LIN {X 0,Y 517.007,Z 176.899,A -85,B 0,C 180,E1 -4953.117,E2 -4953.117} C_VEL
LIN {X 0,Y 517.003,Z 176.9,A -85,B 0,C 180,E1 -4956.243,E2 -4956.243} C_VEL
LIN {X 0,Y 516.949,Z 176.905,A -85,B 0,C 180,E1 -4959.389,E2 -4959.389} C_VEL
LIN {X 0,Y 516.942,Z 176.905,A -85,B 0,C 180,E1 -4961.807,E2 -4961.807} C_VEL
LIN {X 0,Y 516.719,Z 176.937,A -85,B 0,C 180,E1 -4964.171,E2 -4964.171} C_VEL
LIN {X 0,Y 516.698,Z 177.952,A -85,B 0,C 180,E1 -4965.049,E2 -4965.049} C_VEL
LIN {X 0,Y 516.599,Z 183.078,A -85,B 0,C 180,E1 -4968.234,E2 -4968.234} C_VEL
LIN {X 0,Y 516.547,Z 187.118,A -85,B 0,C 180,E1 -4970.717,E2 -4970.717} C_VEL
LIN {X 0,Y 516.494,Z 191.277,A -85,B 0,C 180,E1 -4973.241,E2 -4973.241} C_VEL
LIN {X 0,Y 516.447,Z 196.01,A -85,B 0,C 180,E1 -4976.087,E2 -4976.087} C_VEL
LIN {X 0,Y 516.351,Z 199.966,A -85,B 0,C 180,E1 -4978.449,E2 -4978.449} C_VEL
LIN {X 0,Y 516.31,Z 204.548,A -85,B 0,C 180,E1 -4981.148,E2 -4981.148} C_VEL
LIN {X 0,Y 516.283,Z 209.351,A -85,B 0,C 180,E1 -4983.926,E2 -4983.926} C_VEL
LIN {X 0,Y 516.318,Z 211.119,A -85,B 0,C 180,E1 -4984.972,E2 -4984.972} C_VEL
LIN {X 0,Y 517.437,Z 219.61,A -85,B 0,C 180,E1 -4985.283,E2 -4985.283} C_VEL
LIN {X 0,Y 517.351,Z 228.117,A -85,B 0,C 180,E1 -4985.662,E2 -4985.662} C_VEL
LIN {X 0,Y 517.145,Z 236.097,A -85,B 0,C 180,E1 -4986.119,E2 -4986.119} C_VEL
LIN {X 0,Y 516.974,Z 244.6,A -85,B 0,C 180,E1 -4986.738,E2 -4986.738} C_VEL
LIN {X 0,Y 516.823,Z 252.774,A -85,B 0,C 180,E1 -4987.483,E2 -4987.483} C_VEL
LIN {X 0,Y 516.707,Z 259.834,A -85,B 0,C 180,E1 -4988.297,E2 -4988.297} C_VEL
LIN {X 0,Y 516.566,Z 265.762,A -85,B 0,C 180,E1 -4989.152,E2 -4989.152} C_VEL
LIN {X 0,Y 516.446,Z 270.792,A -85,B 0,C 180,E1 -4990.052,E2 -4990.052} C_VEL
LIN {X 0,Y 516.369,Z 275.581,A -85,B 0,C 180,E1 -4991.159,E2 -4991.159} C_VEL
LIN {X 0,Y 516.287,Z 279.039,A -85,B 0,C 180,E1 -4992.261,E2 -4992.261} C_VEL
LIN {X 0,Y 516.281,Z 280.387,A -85,B 0,C 180,E1 -4992.893,E2 -4992.893} C_VEL
LIN {X 0,Y 516.244,Z 281.973,A -85,B 0,C 180,E1 -4993.971,E2 -4993.971} C_VEL
LIN {X 0,Y 516.246,Z 282.511,A -85,B 0,C 180,E1 -4995.065,E2 -4995.065} C_VEL
LIN {X 0,Y 516.241,Z 281.912,A -85,B 0,C 180,E1 -4996.181,E2 -4996.181} C_VEL
LIN {X 0,Y 516.271,Z 280.176,A -85,B 0,C 180,E1 -4997.316,E2 -4997.316} C_VEL
LIN {X 0,Y 516.325,Z 278.103,A -85,B 0,C 180,E1 -4998.168,E2 -4998.168} C_VEL
LIN {X 0,Y 516.357,Z 274.57,A -85,B 0,C 180,E1 -4999.209,E2 -4999.209} C_VEL
LIN {X 0,Y 516.457,Z 269.892,A -85,B 0,C 180,E1 -5000.241,E2 -5000.241} C_VEL
LIN {X 0,Y 516.592,Z 263.797,A -85,B 0,C 180,E1 -5001.26,E2 -5001.26} C_VEL
LIN {X 0,Y 516.704,Z 257.558,A -85,B 0,C 180,E1 -5002.082,E2 -5002.082} C_VEL
LIN {X 0,Y 516.85,Z 251.253,A -85,B 0,C 180,E1 -5002.765,E2 -5002.765} C_VEL
LIN {X 0,Y 516.992,Z 244.179,A -85,B 0,C 180,E1 -5003.397,E2 -5003.397} C_VEL
LIN {X 0,Y 517.156,Z 235.77,A -85,B 0,C 180,E1 -5004.003,E2 -5004.003} C_VEL
LIN {X 0,Y 517.368,Z 225.06,A -85,B 0,C 180,E1 -5004.592,E2 -5004.592} C_VEL
LIN {X 0,Y 517.228,Z 217.017,A -85,B 0,C 180,E1 -5004.918,E2 -5004.918} C_VEL
LIN {X 0,Y 516.323,Z 211.255,A -85,B 0,C 180,E1 -5005.133,E2 -5005.133} C_VEL
LIN {X 0,Y 516.328,Z 206.51,A -85,B 0,C 180,E1 -5007.938,E2 -5007.938} C_VEL
LIN {X 0,Y 516.368,Z 201.944,A -85,B 0,C 180,E1 -5010.662,E2 -5010.662} C_VEL
LIN {X 0,Y 516.441,Z 197.541,A -85,B 0,C 180,E1 -5013.316,E2 -5013.316} C_VEL
LIN {X 0,Y 516.509,Z 193.252,A -85,B 0,C 180,E1 -5015.909,E2 -5015.909} C_VEL
LIN {X 0,Y 516.551,Z 189.113,A -85,B 0,C 180,E1 -5018.449,E2 -5018.449} C_VEL
LIN {X 0,Y 516.616,Z 185.061,A -85,B 0,C 180,E1 -5020.945,E2 -5020.945} C_VEL
LIN {X 0,Y 516.71,Z 181.143,A -85,B 0,C 180,E1 -5023.404,E2 -5023.404} C_VEL
LIN {X 0,Y 516.726,Z 177.242,A -85,B 0,C 180,E1 -5025.83,E2 -5025.83} C_VEL
LIN {X 0,Y 516.889,Z 176.918,A -85,B 0,C 180,E1 -5027.436,E2 -5027.436} C_VEL
LIN {X 0,Y 516.906,Z 176.913,A -85,B 0,C 180,E1 -5029.82,E2 -5029.82} C_VEL
LIN {X 0,Y 516.979,Z 176.906,A -85,B 0,C 180,E1 -5032.188,E2 -5032.188} C_VEL
LIN {X 0,Y 517.03,Z 176.9,A -85,B 0,C 180,E1 -5034.541,E2 -5034.541} C_VEL
LIN {X 0,Y 517.085,Z 176.89,A -85,B 0,C 180,E1 -5037.664,E2 -5037.664} C_VEL
LIN {X 0,Y 517.097,Z 176.887,A -85,B 0,C 180,E1 -5040.779,E2 -5040.779} C_VEL
LIN {X 0,Y 517.013,Z 176.897,A -85,B 0,C 180,E1 -5043.118,E2 -5043.118} C_VEL
LIN {X 0,Y 517.013,Z 176.898,A -85,B 0,C 180,E1 -5046.244,E2 -5046.244} C_VEL
LIN {X 0,Y 516.951,Z 176.908,A -85,B 0,C 180,E1 -5049.39,E2 -5049.39} C_VEL
LIN {X 0,Y 516.955,Z 176.906,A -85,B 0,C 180,E1 -5051.808,E2 -5051.808} C_VEL
LIN {X 0,Y 516.947,Z 176.908,A -85,B 0,C 180,E1 -5055.147,E2 -5055.147} C_VEL
LIN {X 0,Y 516.928,Z 176.908,A -85,B 0,C 180,E1 -5058.223,E2 -5058.223} C_VEL
LIN {X 0,Y 516.915,Z 176.911,A -85,B 0,C 180,E1 -5060.702,E2 -5060.702} C_VEL
LIN {X 0,Y 516.894,Z 176.913,A -85,B 0,C 180,E1 -5064.073,E2 -5064.073} C_VEL
LIN {X 0,Y 516.926,Z 176.91,A -85,B 0,C 180,E1 -5066.658,E2 -5066.658} C_VEL
LIN {X 0,Y 516.914,Z 176.91,A -85,B 0,C 180,E1 -5069.524,E2 -5069.524} C_VEL
LIN {X 0,Y 516.9,Z 176.912,A -85,B 0,C 180,E1 -5072.544,E2 -5072.544} C_VEL
LIN {X 0,Y 516.869,Z 176.915,A -85,B 0,C 180,E1 -5075.33,E2 -5075.33} C_VEL
LIN {X 0,Y 516.882,Z 176.916,A -85,B 0,C 180,E1 -5077.943,E2 -5077.943} C_VEL
LIN {X 0,Y 516.885,Z 176.914,A -85,B 0,C 180,E1 -5080.742,E2 -5080.742} C_VEL
LIN {X 0,Y 516.886,Z 176.916,A -85,B 0,C 180,E1 -5082.832,E2 -5082.832} C_VEL
LIN {X 0,Y 516.925,Z 176.912,A -85,B 0,C 180,E1 -5085.01,E2 -5085.01} C_VEL
LIN {X 0,Y 516.915,Z 176.913,A -85,B 0,C 180,E1 -5088.399,E2 -5088.399} C_VEL
LIN {X 0,Y 516.882,Z 176.914,A -85,B 0,C 180,E1 -5091.284,E2 -5091.284} C_VEL
LIN {X 0,Y 516.889,Z 176.919,A -85,B 0,C 180,E1 -5094.221,E2 -5094.221} C_VEL
LIN {X 0,Y 516.936,Z 177.011,A -85,B 0,C 180,E1 -5096.998,E2 -5096.998} C_VEL
LIN {X 0,Y 517.781,Z 182.254,A -85,B 0,C 180,E1 -5098.95,E2 -5098.95} C_VEL
LIN {X 0,Y 517.707,Z 187.477,A -85,B 0,C 180,E1 -5100.744,E2 -5100.744} C_VEL
LIN {X 0,Y 517.327,Z 196.482,A -85,B 0,C 180,E1 -5103.718,E2 -5103.718} C_VEL
LIN {X 0,Y 517.076,Z 204.771,A -85,B 0,C 180,E1 -5106.362,E2 -5106.362} C_VEL
LIN {X 0,Y 516.906,Z 214.303,A -85,B 0,C 180,E1 -5109.298,E2 -5109.298} C_VEL
LIN {X 0,Y 516.744,Z 223.934,A -85,B 0,C 180,E1 -5112.183,E2 -5112.183} C_VEL
LIN {X 0,Y 516.556,Z 235.008,A -85,B 0,C 180,E1 -5115.422,E2 -5115.422} C_VEL
LIN {X 0,Y 516.483,Z 245.506,A -85,B 0,C 180,E1 -5118.446,E2 -5118.446} C_VEL
LIN {X 0,Y 516.443,Z 247.582,A -85,B 0,C 180,E1 -5119.042,E2 -5119.042} C_VEL
LIN {X 0,Y 517.53,Z 258.934,A -85,B 0,C 180,E1 -5119.387,E2 -5119.387} C_VEL
LIN {X 0,Y 517.335,Z 269.543,A -85,B 0,C 180,E1 -5119.828,E2 -5119.828} C_VEL
LIN {X 0,Y 517.156,Z 278.389,A -85,B 0,C 180,E1 -5120.319,E2 -5120.319} C_VEL
LIN {X 0,Y 516.972,Z 286.814,A -85,B 0,C 180,E1 -5120.907,E2 -5120.907} C_VEL
LIN {X 0,Y 516.814,Z 294.777,A -85,B 0,C 180,E1 -5121.594,E2 -5121.594} C_VEL
LIN {X 0,Y 516.652,Z 302.217,A -85,B 0,C 180,E1 -5122.379,E2 -5122.379} C_VEL
LIN {X 0,Y 516.54,Z 309.564,A -85,B 0,C 180,E1 -5123.331,E2 -5123.331} C_VEL
LIN {X 0,Y 516.437,Z 315.695,A -85,B 0,C 180,E1 -5124.338,E2 -5124.338} C_VEL
LIN {X 0,Y 516.309,Z 320.354,A -85,B 0,C 180,E1 -5125.315,E2 -5125.315} C_VEL
LIN {X 0,Y 516.361,Z 323.384,A -85,B 0,C 180,E1 -5126.098,E2 -5126.098} C_VEL
LIN {X 0,Y 516.293,Z 325.728,A -85,B 0,C 180,E1 -5126.879,E2 -5126.879} C_VEL
LIN {X 0,Y 516.263,Z 327.495,A -85,B 0,C 180,E1 -5127.66,E2 -5127.66} C_VEL
LIN {X 0,Y 516.191,Z 328.76,A -85,B 0,C 180,E1 -5128.44,E2 -5128.44} C_VEL
LIN {X 0,Y 516.164,Z 329.55,A -85,B 0,C 180,E1 -5129.22,E2 -5129.22} C_VEL
LIN {X 0,Y 516.165,Z 329.852,A -85,B 0,C 180,E1 -5130,E2 -5130} C_VEL
LIN {X 0,Y 516.164,Z 329.558,A -85,B 0,C 180,E1 -5130.78,E2 -5130.78} C_VEL
LIN {X 0,Y 516.191,Z 328.774,A -85,B 0,C 180,E1 -5131.561,E2 -5131.561} C_VEL
LIN {X 0,Y 516.263,Z 327.515,A -85,B 0,C 180,E1 -5132.341,E2 -5132.341} C_VEL
LIN {X 0,Y 516.323,Z 324.596,A -85,B 0,C 180,E1 -5133.512,E2 -5133.512} C_VEL
LIN {X 0,Y 516.339,Z 321.929,A -85,B 0,C 180,E1 -5134.293,E2 -5134.293} C_VEL
LIN {X 0,Y 516.421,Z 316.716,A -85,B 0,C 180,E1 -5135.467,E2 -5135.467} C_VEL
LIN {X 0,Y 516.515,Z 309.801,A -85,B 0,C 180,E1 -5136.645,E2 -5136.645} C_VEL
LIN {X 0,Y 516.654,Z 302.305,A -85,B 0,C 180,E1 -5137.622,E2 -5137.622} C_VEL
LIN {X 0,Y 516.815,Z 294.884,A -85,B 0,C 180,E1 -5138.406,E2 -5138.406} C_VEL
LIN {X 0,Y 516.974,Z 286.932,A -85,B 0,C 180,E1 -5139.093,E2 -5139.093} C_VEL
LIN {X 0,Y 517.186,Z 277.013,A -85,B 0,C 180,E1 -5139.78,E2 -5139.78} C_VEL
LIN {X 0,Y 517.414,Z 266.525,A -85,B 0,C 180,E1 -5140.319,E2 -5140.319} C_VEL
LIN {X 0,Y 517.41,Z 257.056,A -85,B 0,C 180,E1 -5140.678,E2 -5140.678} C_VEL
LIN {X 0,Y 516.444,Z 247.771,A -85,B 0,C 180,E1 -5140.958,E2 -5140.958} C_VEL
LIN {X 0,Y 516.573,Z 236.715,A -85,B 0,C 180,E1 -5144.176,E2 -5144.176} C_VEL
LIN {X 0,Y 516.718,Z 225.681,A -85,B 0,C 180,E1 -5147.411,E2 -5147.411} C_VEL
LIN {X 0,Y 516.927,Z 214.606,A -85,B 0,C 180,E1 -5150.701,E2 -5150.701} C_VEL
LIN {X 0,Y 517.1,Z 205.055,A -85,B 0,C 180,E1 -5153.637,E2 -5153.637} C_VEL
LIN {X 0,Y 517.415,Z 195.575,A -85,B 0,C 180,E1 -5156.631,E2 -5156.631} C_VEL
LIN {X 0,Y 517.767,Z 186.175,A -85,B 0,C 180,E1 -5159.69,E2 -5159.69} C_VEL
LIN {X 0,Y 517.717,Z 181.674,A -85,B 0,C 180,E1 -5161.215,E2 -5161.215} C_VEL
LIN {X 0,Y 516.92,Z 176.911,A -85,B 0,C 180,E1 -5162.945,E2 -5162.945} C_VEL
LIN {X 0,Y 516.874,Z 176.914,A -85,B 0,C 180,E1 -5165.78,E2 -5165.78} C_VEL
LIN {X 0,Y 516.884,Z 176.914,A -85,B 0,C 180,E1 -5168.716,E2 -5168.716} C_VEL
LIN {X 0,Y 516.915,Z 176.911,A -85,B 0,C 180,E1 -5171.775,E2 -5171.775} C_VEL
LIN {X 0,Y 516.899,Z 176.911,A -85,B 0,C 180,E1 -5175.007,E2 -5175.007} C_VEL
LIN {X 0,Y 516.914,Z 176.91,A -85,B 0,C 180,E1 -5178.399,E2 -5178.399} C_VEL
LIN {X 0,Y 516.883,Z 176.912,A -85,B 0,C 180,E1 -5181.284,E2 -5181.284} C_VEL
LIN {X 0,Y 516.875,Z 176.916,A -85,B 0,C 180,E1 -5184.22,E2 -5184.22} C_VEL
LIN {X 0,Y 516.899,Z 176.913,A -85,B 0,C 180,E1 -5187.053,E2 -5187.053} C_VEL
LIN {X 0,Y 516.896,Z 176.913,A -85,B 0,C 180,E1 -5189.796,E2 -5189.796} C_VEL
LIN {X 0,Y 516.927,Z 176.907,A -85,B 0,C 180,E1 -5192.467,E2 -5192.467} C_VEL
LIN {X 0,Y 516.88,Z 176.914,A -85,B 0,C 180,E1 -5195.07,E2 -5195.07} C_VEL
LIN {X 0,Y 516.874,Z 176.915,A -85,B 0,C 180,E1 -5197.621,E2 -5197.621} C_VEL
LIN {X 0,Y 516.936,Z 176.907,A -85,B 0,C 180,E1 -5200.13,E2 -5200.13} C_VEL
LIN {X 0,Y 516.911,Z 176.91,A -85,B 0,C 180,E1 -5202.595,E2 -5202.595} C_VEL
LIN {X 0,Y 516.948,Z 176.908,A -85,B 0,C 180,E1 -5205.03,E2 -5205.03} C_VEL
LIN {X 0,Y 516.971,Z 176.902,A -85,B 0,C 180,E1 -5208.233,E2 -5208.233} C_VEL
LIN {X 0,Y 516.959,Z 176.906,A -85,B 0,C 180,E1 -5211.399,E2 -5211.399} C_VEL
LIN {X 0,Y 517.003,Z 176.901,A -85,B 0,C 180,E1 -5213.756,E2 -5213.756} C_VEL
LIN {X 0,Y 517.013,Z 176.897,A -85,B 0,C 180,E1 -5216.882,E2 -5216.882} C_VEL
LIN {X 0,Y 517.09,Z 176.889,A -85,B 0,C 180,E1 -5219.999,E2 -5219.999} C_VEL
LIN {X 0,Y 517.016,Z 176.897,A -85,B 0,C 180,E1 -5223.116,E2 -5223.116} C_VEL
LIN {X 0,Y 517.005,Z 176.897,A -85,B 0,C 180,E1 -5226.242,E2 -5226.242} C_VEL
LIN {X 0,Y 516.944,Z 176.906,A -85,B 0,C 180,E1 -5229.389,E2 -5229.389} C_VEL
LIN {X 0,Y 516.955,Z 176.905,A -85,B 0,C 180,E1 -5231.806,E2 -5231.806} C_VEL
LIN {X 0,Y 516.947,Z 176.906,A -85,B 0,C 180,E1 -5235.146,E2 -5235.146} C_VEL
LIN {X 0,Y 516.918,Z 176.911,A -85,B 0,C 180,E1 -5238.222,E2 -5238.222} C_VEL
LIN {X 0,Y 516.913,Z 176.912,A -85,B 0,C 180,E1 -5240.701,E2 -5240.701} C_VEL
LIN {X 0,Y 516.891,Z 176.912,A -85,B 0,C 180,E1 -5244.072,E2 -5244.072} C_VEL
LIN {X 0,Y 516.926,Z 176.909,A -85,B 0,C 180,E1 -5246.657,E2 -5246.657} C_VEL
LIN {X 0,Y 516.91,Z 176.911,A -85,B 0,C 180,E1 -5249.523,E2 -5249.523} C_VEL
LIN {X 0,Y 516.896,Z 176.912,A -85,B 0,C 180,E1 -5252.543,E2 -5252.543} C_VEL
LIN {X 0,Y 516.879,Z 176.912,A -85,B 0,C 180,E1 -5255.331,E2 -5255.331} C_VEL
LIN {X 0,Y 516.877,Z 176.914,A -85,B 0,C 180,E1 -5257.942,E2 -5257.942} C_VEL
LIN {X 0,Y 516.881,Z 176.914,A -85,B 0,C 180,E1 -5260.741,E2 -5260.741} C_VEL
LIN {X 0,Y 516.879,Z 176.912,A -85,B 0,C 180,E1 -5262.83,E2 -5262.83} C_VEL
LIN {X 0,Y 516.918,Z 176.91,A -85,B 0,C 180,E1 -5265.009,E2 -5265.009} C_VEL
LIN {X 0,Y 516.912,Z 176.911,A -85,B 0,C 180,E1 -5268.397,E2 -5268.397} C_VEL
LIN {X 0,Y 516.876,Z 176.914,A -85,B 0,C 180,E1 -5270.298,E2 -5270.298} C_VEL
LIN {X 0,Y 516.205,Z 176.998,A -85,B 0,C 180,E1 -5270.948,E2 -5270.948} C_VEL
LIN {X 0,Y 513.36,Z 177.354,A -85,B 0,C 180,E1 -5272.003,E2 -5272.003} C_VEL
LIN {X 0,Y 510.954,Z 177.656,A -85,B 0,C 180,E1 -5272.854,E2 -5272.854} C_VEL
LIN {X 0,Y 509.914,Z 177.784,A -85,B 0,C 180,E1 -5273.51,E2 -5273.51} C_VEL
LIN {X 0,Y 509.826,Z 177.793,A -85,B 0,C 180,E1 -5273.733,E2 -5273.733} C_VEL
LIN {X 0,Y 509.858,Z 177.789,A -85,B 0,C 180,E1 -5276.539,E2 -5276.539} C_VEL
LIN {X 0,Y 509.845,Z 177.791,A -85,B 0,C 180,E1 -5279.334,E2 -5279.334} C_VEL
LIN {X 0,Y 509.888,Z 177.784,A -85,B 0,C 180,E1 -5282.054,E2 -5282.054} C_VEL
LIN {X 0,Y 509.87,Z 177.786,A -85,B 0,C 180,E1 -5284.703,E2 -5284.703} C_VEL
LIN {X 0,Y 509.829,Z 177.793,A -85,B 0,C 180,E1 -5287.454,E2 -5287.454} C_VEL
LIN {X 0,Y 509.909,Z 177.782,A -85,B 0,C 180,E1 -5289.844,E2 -5289.844} C_VEL
LIN {X 0,Y 509.877,Z 177.788,A -85,B 0,C 180,E1 -5293.174,E2 -5293.174} C_VEL
LIN {X 0,Y 509.866,Z 177.788,A -85,B 0,C 180,E1 -5295.634,E2 -5295.634} C_VEL
LIN {X 0,Y 509.913,Z 177.782,A -85,B 0,C 180,E1 -5298.874,E2 -5298.874} C_VEL
LIN {X 0,Y 509.943,Z 177.779,A -85,B 0,C 180,E1 -5302.078,E2 -5302.078} C_VEL
LIN {X 0,Y 509.975,Z 177.776,A -85,B 0,C 180,E1 -5304.464,E2 -5304.464} C_VEL
LIN {X 0,Y 510.044,Z 177.764,A -85,B 0,C 180,E1 -5307.631,E2 -5307.631} C_VEL
LIN {X 0,Y 510.044,Z 177.765,A -85,B 0,C 180,E1 -5310,E2 -5310} C_VEL
LIN {X 0,Y 510.048,Z 177.766,A -85,B 0,C 180,E1 -5312.369,E2 -5312.369} C_VEL
LIN {X 0,Y 509.971,Z 177.775,A -85,B 0,C 180,E1 -5316.33,E2 -5316.33} C_VEL
LIN {X 0,Y 509.909,Z 177.783,A -85,B 0,C 180,E1 -5318.72,E2 -5318.72} C_VEL
LIN {X 0,Y 509.893,Z 177.784,A -85,B 0,C 180,E1 -5321.932,E2 -5321.932} C_VEL
LIN {X 0,Y 509.648,Z 177.818,A -85,B 0,C 180,E1 -5324.372,E2 -5324.372} C_VEL
LIN {X 0,Y 509.562,Z 181.569,A -85,B 0,C 180,E1 -5326.836,E2 -5326.836} C_VEL
LIN {X 0,Y 509.507,Z 185.566,A -85,B 0,C 180,E1 -5329.332,E2 -5329.332} C_VEL
LIN {X 0,Y 509.466,Z 190.606,A -85,B 0,C 180,E1 -5332.447,E2 -5332.447} C_VEL
LIN {X 0,Y 509.385,Z 195.348,A -85,B 0,C 180,E1 -5335.322,E2 -5335.322} C_VEL
LIN {X 0,Y 509.314,Z 199.766,A -85,B 0,C 180,E1 -5337.98,E2 -5337.98} C_VEL
LIN {X 0,Y 509.228,Z 205.106,A -85,B 0,C 180,E1 -5341.167,E2 -5341.167} C_VEL
LIN {X 0,Y 509.21,Z 210.109,A -85,B 0,C 180,E1 -5344.097,E2 -5344.097} C_VEL
LIN {X 0,Y 509.219,Z 211.361,A -85,B 0,C 180,E1 -5344.823,E2 -5344.823} C_VEL
LIN {X 0,Y 510.43,Z 220.001,A -85,B 0,C 180,E1 -5345.149,E2 -5345.149} C_VEL
LIN {X 0,Y 510.323,Z 229.555,A -85,B 0,C 180,E1 -5345.591,E2 -5345.591} C_VEL
LIN {X 0,Y 510.132,Z 238.671,A -85,B 0,C 180,E1 -5346.147,E2 -5346.147} C_VEL
LIN {X 0,Y 509.922,Z 248.487,A -85,B 0,C 180,E1 -5346.931,E2 -5346.931} C_VEL
LIN {X 0,Y 509.724,Z 256.142,A -85,B 0,C 180,E1 -5347.722,E2 -5347.722} C_VEL
LIN {X 0,Y 509.616,Z 261.255,A -85,B 0,C 180,E1 -5348.359,E2 -5348.359} C_VEL
LIN {X 0,Y 509.515,Z 266.414,A -85,B 0,C 180,E1 -5349.128,E2 -5349.128} C_VEL
LIN {X 0,Y 509.396,Z 270.74,A -85,B 0,C 180,E1 -5349.907,E2 -5349.907} C_VEL
LIN {X 0,Y 509.291,Z 274.075,A -85,B 0,C 180,E1 -5350.628,E2 -5350.628} C_VEL
LIN {X 0,Y 509.238,Z 278.205,A -85,B 0,C 180,E1 -5351.821,E2 -5351.821} C_VEL
LIN {X 0,Y 509.201,Z 280.965,A -85,B 0,C 180,E1 -5352.989,E2 -5352.989} C_VEL
LIN {X 0,Y 509.151,Z 282.47,A -85,B 0,C 180,E1 -5354.13,E2 -5354.13} C_VEL
LIN {X 0,Y 509.15,Z 282.779,A -85,B 0,C 180,E1 -5355.255,E2 -5355.255} C_VEL
LIN {X 0,Y 509.167,Z 282.042,A -85,B 0,C 180,E1 -5356.36,E2 -5356.36} C_VEL
LIN {X 0,Y 509.183,Z 280.308,A -85,B 0,C 180,E1 -5357.444,E2 -5357.444} C_VEL
LIN {X 0,Y 509.26,Z 277.551,A -85,B 0,C 180,E1 -5358.517,E2 -5358.517} C_VEL
LIN {X 0,Y 509.321,Z 273.734,A -85,B 0,C 180,E1 -5359.57,E2 -5359.57} C_VEL
LIN {X 0,Y 509.463,Z 268.582,A -85,B 0,C 180,E1 -5360.614,E2 -5360.614} C_VEL
LIN {X 0,Y 509.556,Z 263.852,A -85,B 0,C 180,E1 -5361.385,E2 -5361.385} C_VEL
LIN {X 0,Y 509.71,Z 257.05,A -85,B 0,C 180,E1 -5362.278,E2 -5362.278} C_VEL
LIN {X 0,Y 509.845,Z 251.266,A -85,B 0,C 180,E1 -5362.904,E2 -5362.904} C_VEL
LIN {X 0,Y 510.012,Z 243.965,A -85,B 0,C 180,E1 -5363.558,E2 -5363.558} C_VEL
LIN {X 0,Y 510.169,Z 235.815,A -85,B 0,C 180,E1 -5364.148,E2 -5364.148} C_VEL
LIN {X 0,Y 510.388,Z 225.346,A -85,B 0,C 180,E1 -5364.728,E2 -5364.728} C_VEL
LIN {X 0,Y 510.327,Z 218.252,A -85,B 0,C 180,E1 -5365.025,E2 -5365.025} C_VEL
LIN {X 0,Y 509.244,Z 211.567,A -85,B 0,C 180,E1 -5365.271,E2 -5365.271} C_VEL
LIN {X 0,Y 509.255,Z 206.375,A -85,B 0,C 180,E1 -5368.372,E2 -5368.372} C_VEL
LIN {X 0,Y 509.305,Z 201.796,A -85,B 0,C 180,E1 -5371.121,E2 -5371.121} C_VEL
LIN {X 0,Y 509.405,Z 197.384,A -85,B 0,C 180,E1 -5373.802,E2 -5373.802} C_VEL
LIN {X 0,Y 509.434,Z 193.145,A -85,B 0,C 180,E1 -5376.418,E2 -5376.418} C_VEL
LIN {X 0,Y 509.483,Z 188.986,A -85,B 0,C 180,E1 -5378.983,E2 -5378.983} C_VEL
LIN {X 0,Y 509.62,Z 184.064,A -85,B 0,C 180,E1 -5382.093,E2 -5382.093} C_VEL
LIN {X 0,Y 509.677,Z 179.641,A -85,B 0,C 180,E1 -5384.849,E2 -5384.849} C_VEL
LIN {X 0,Y 509.691,Z 178.416,A -85,B 0,C 180,E1 -5385.63,E2 -5385.63} C_VEL
LIN {X 0,Y 509.743,Z 177.808,A -85,B 0,C 180,E1 -5386.445,E2 -5386.445} C_VEL
LIN {X 0,Y 509.912,Z 177.785,A -85,B 0,C 180,E1 -5388.875,E2 -5388.875} C_VEL
LIN {X 0,Y 509.952,Z 177.781,A -85,B 0,C 180,E1 -5392.079,E2 -5392.079} C_VEL
LIN {X 0,Y 509.982,Z 177.778,A -85,B 0,C 180,E1 -5394.465,E2 -5394.465} C_VEL
LIN {X 0,Y 510.056,Z 177.766,A -85,B 0,C 180,E1 -5397.632,E2 -5397.632} C_VEL
LIN {X 0,Y 510.067,Z 177.762,A -85,B 0,C 180,E1 -5400.79,E2 -5400.79} C_VEL
LIN {X 0,Y 509.955,Z 177.776,A -85,B 0,C 180,E1 -5403.161,E2 -5403.161} C_VEL
LIN {X 0,Y 509.981,Z 177.774,A -85,B 0,C 180,E1 -5406.33,E2 -5406.33} C_VEL
LIN {X 0,Y 509.892,Z 177.786,A -85,B 0,C 180,E1 -5409.521,E2 -5409.521} C_VEL
LIN {X 0,Y 509.907,Z 177.783,A -85,B 0,C 180,E1 -5411.932,E2 -5411.932} C_VEL
LIN {X 0,Y 509.897,Z 177.786,A -85,B 0,C 180,E1 -5415.242,E2 -5415.242} C_VEL
LIN {X 0,Y 509.892,Z 177.784,A -85,B 0,C 180,E1 -5418.001,E2 -5418.001} C_VEL
LIN {X 0,Y 509.853,Z 177.791,A -85,B 0,C 180,E1 -5421.002,E2 -5421.002} C_VEL
LIN {X 0,Y 509.825,Z 177.793,A -85,B 0,C 180,E1 -5423.564,E2 -5423.564} C_VEL
LIN {X 0,Y 509.914,Z 177.782,A -85,B 0,C 180,E1 -5426.379,E2 -5426.379} C_VEL
LIN {X 0,Y 509.879,Z 177.788,A -85,B 0,C 180,E1 -5428.845,E2 -5428.845} C_VEL
LIN {X 0,Y 509.824,Z 177.793,A -85,B 0,C 180,E1 -5431.59,E2 -5431.59} C_VEL
LIN {X 0,Y 509.85,Z 177.791,A -85,B 0,C 180,E1 -5434.414,E2 -5434.414} C_VEL
LIN {X 0,Y 509.818,Z 177.793,A -85,B 0,C 180,E1 -5437.341,E2 -5437.341} C_VEL
LIN {X 0,Y 509.84,Z 177.794,A -85,B 0,C 180,E1 -5440.382,E2 -5440.382} C_VEL
LIN {X 0,Y 509.826,Z 177.794,A -85,B 0,C 180,E1 -5443.062,E2 -5443.062} C_VEL
LIN {X 0,Y 509.832,Z 177.794,A -85,B 0,C 180,E1 -5445.793,E2 -5445.793} C_VEL
LIN {X 0,Y 509.857,Z 177.791,A -85,B 0,C 180,E1 -5448.575,E2 -5448.575} C_VEL
LIN {X 0,Y 509.853,Z 177.792,A -85,B 0,C 180,E1 -5451.787,E2 -5451.787} C_VEL
LIN {X 0,Y 509.844,Z 177.796,A -85,B 0,C 180,E1 -5454.623,E2 -5454.623} C_VEL
LIN {X 0,Y 509.901,Z 177.948,A -85,B 0,C 180,E1 -5456.813,E2 -5456.813} C_VEL
LIN {X 0,Y 510.809,Z 183.697,A -85,B 0,C 180,E1 -5458.984,E2 -5458.984} C_VEL
LIN {X 0,Y 510.651,Z 190.097,A -85,B 0,C 180,E1 -5461.204,E2 -5461.204} C_VEL
LIN {X 0,Y 510.243,Z 199.29,A -85,B 0,C 180,E1 -5464.286,E2 -5464.286} C_VEL
LIN {X 0,Y 510.016,Z 207.349,A -85,B 0,C 180,E1 -5466.876,E2 -5466.876} C_VEL
LIN {X 0,Y 509.773,Z 216.843,A -85,B 0,C 180,E1 -5469.839,E2 -5469.839} C_VEL
LIN {X 0,Y 509.61,Z 226.462,A -85,B 0,C 180,E1 -5472.752,E2 -5472.752} C_VEL
LIN {X 0,Y 509.447,Z 236.097,A -85,B 0,C 180,E1 -5475.622,E2 -5475.622} C_VEL
LIN {X 0,Y 509.395,Z 247.354,A -85,B 0,C 180,E1 -5478.914,E2 -5478.914} C_VEL
LIN {X 0,Y 510.481,Z 258.417,A -85,B 0,C 180,E1 -5479.239,E2 -5479.239} C_VEL
LIN {X 0,Y 510.328,Z 269.108,A -85,B 0,C 180,E1 -5479.687,E2 -5479.687} C_VEL
LIN {X 0,Y 510.132,Z 277.976,A -85,B 0,C 180,E1 -5480.184,E2 -5480.184} C_VEL
LIN {X 0,Y 509.957,Z 286.419,A -85,B 0,C 180,E1 -5480.781,E2 -5480.781} C_VEL
LIN {X 0,Y 509.771,Z 294.396,A -85,B 0,C 180,E1 -5481.477,E2 -5481.477} C_VEL
LIN {X 0,Y 509.584,Z 301.846,A -85,B 0,C 180,E1 -5482.272,E2 -5482.272} C_VEL
LIN {X 0,Y 509.466,Z 308.243,A -85,B 0,C 180,E1 -5483.105,E2 -5483.105} C_VEL
LIN {X 0,Y 509.369,Z 315.348,A -85,B 0,C 180,E1 -5484.259,E2 -5484.259} C_VEL
LIN {X 0,Y 509.223,Z 320.013,A -85,B 0,C 180,E1 -5485.25,E2 -5485.25} C_VEL
LIN {X 0,Y 509.258,Z 323.046,A -85,B 0,C 180,E1 -5486.043,E2 -5486.043} C_VEL
LIN {X 0,Y 509.211,Z 325.394,A -85,B 0,C 180,E1 -5486.835,E2 -5486.835} C_VEL
LIN {X 0,Y 509.191,Z 327.166,A -85,B 0,C 180,E1 -5487.627,E2 -5487.627} C_VEL
LIN {X 0,Y 509.111,Z 328.432,A -85,B 0,C 180,E1 -5488.418,E2 -5488.418} C_VEL
LIN {X 0,Y 509.077,Z 329.224,A -85,B 0,C 180,E1 -5489.209,E2 -5489.209} C_VEL
LIN {X 0,Y 509.076,Z 329.527,A -85,B 0,C 180,E1 -5490,E2 -5490} C_VEL
LIN {X 0,Y 509.077,Z 329.235,A -85,B 0,C 180,E1 -5490.791,E2 -5490.791} C_VEL
LIN {X 0,Y 509.111,Z 328.451,A -85,B 0,C 180,E1 -5491.582,E2 -5491.582} C_VEL
LIN {X 0,Y 509.192,Z 327.191,A -85,B 0,C 180,E1 -5492.373,E2 -5492.373} C_VEL
LIN {X 0,Y 509.243,Z 324.271,A -85,B 0,C 180,E1 -5493.561,E2 -5493.561} C_VEL
LIN {X 0,Y 509.234,Z 321.599,A -85,B 0,C 180,E1 -5494.353,E2 -5494.353} C_VEL
LIN {X 0,Y 509.336,Z 316.385,A -85,B 0,C 180,E1 -5495.543,E2 -5495.543} C_VEL
LIN {X 0,Y 509.412,Z 310.259,A -85,B 0,C 180,E1 -5496.619,E2 -5496.619} C_VEL
LIN {X 0,Y 509.548,Z 303.667,A -85,B 0,C 180,E1 -5497.529,E2 -5497.529} C_VEL
LIN {X 0,Y 509.742,Z 295.552,A -85,B 0,C 180,E1 -5498.424,E2 -5498.424} C_VEL
LIN {X 0,Y 509.905,Z 287.798,A -85,B 0,C 180,E1 -5499.12,E2 -5499.12} C_VEL
LIN {X 0,Y 510.102,Z 279.641,A -85,B 0,C 180,E1 -5499.717,E2 -5499.717} C_VEL
LIN {X 0,Y 510.277,Z 271.164,A -85,B 0,C 180,E1 -5500.214,E2 -5500.214} C_VEL
LIN {X 0,Y 510.507,Z 261.264,A -85,B 0,C 180,E1 -5500.661,E2 -5500.661} C_VEL
LIN {X 0,Y 510.171,Z 255.316,A -85,B 0,C 180,E1 -5500.869,E2 -5500.869} C_VEL
LIN {X 0,Y 509.378,Z 247.486,A -85,B 0,C 180,E1 -5501.112,E2 -5501.112} C_VEL
LIN {X 0,Y 509.48,Z 236.424,A -85,B 0,C 180,E1 -5504.377,E2 -5504.377} C_VEL
LIN {X 0,Y 509.644,Z 226.77,A -85,B 0,C 180,E1 -5507.247,E2 -5507.247} C_VEL
LIN {X 0,Y 509.827,Z 216.453,A -85,B 0,C 180,E1 -5510.383,E2 -5510.383} C_VEL
LIN {X 0,Y 510.071,Z 206.308,A -85,B 0,C 180,E1 -5513.552,E2 -5513.552} C_VEL
LIN {X 0,Y 510.331,Z 198.162,A -85,B 0,C 180,E1 -5516.148,E2 -5516.148} C_VEL
LIN {X 0,Y 510.697,Z 188.759,A -85,B 0,C 180,E1 -5519.245,E2 -5519.245} C_VEL
LIN {X 0,Y 510.799,Z 183.569,A -85,B 0,C 180,E1 -5521.012,E2 -5521.012} C_VEL
LIN {X 0,Y 509.885,Z 177.788,A -85,B 0,C 180,E1 -5523.135,E2 -5523.135} C_VEL
LIN {X 0,Y 509.828,Z 177.794,A -85,B 0,C 180,E1 -5526.353,E2 -5526.353} C_VEL
LIN {X 0,Y 509.849,Z 177.791,A -85,B 0,C 180,E1 -5529.353,E2 -5529.353} C_VEL
LIN {X 0,Y 509.836,Z 177.791,A -85,B 0,C 180,E1 -5532.49,E2 -5532.49} C_VEL
LIN {X 0,Y 509.842,Z 177.791,A -85,B 0,C 180,E1 -5535.33,E2 -5535.33} C_VEL
LIN {X 0,Y 509.856,Z 177.789,A -85,B 0,C 180,E1 -5538.574,E2 -5538.574} C_VEL
LIN {X 0,Y 509.854,Z 177.79,A -85,B 0,C 180,E1 -5541.787,E2 -5541.787} C_VEL
LIN {X 0,Y 509.834,Z 177.792,A -85,B 0,C 180,E1 -5544.622,E2 -5544.622} C_VEL
LIN {X 0,Y 509.866,Z 177.787,A -85,B 0,C 180,E1 -5547.481,E2 -5547.481} C_VEL
LIN {X 0,Y 509.863,Z 177.788,A -85,B 0,C 180,E1 -5550.274,E2 -5550.274} C_VEL
LIN {X 0,Y 509.886,Z 177.784,A -85,B 0,C 180,E1 -5552.944,E2 -5552.944} C_VEL
LIN {X 0,Y 509.855,Z 177.789,A -85,B 0,C 180,E1 -5555.573,E2 -5555.573} C_VEL
LIN {X 0,Y 509.827,Z 177.793,A -85,B 0,C 180,E1 -5558.148,E2 -5558.148} C_VEL
LIN {X 0,Y 509.867,Z 177.787,A -85,B 0,C 180,E1 -5560.681,E2 -5560.681} C_VEL
LIN {X 0,Y 509.877,Z 177.786,A -85,B 0,C 180,E1 -5563.174,E2 -5563.174} C_VEL
LIN {X 0,Y 509.868,Z 177.787,A -85,B 0,C 180,E1 -5565.634,E2 -5565.634} C_VEL
LIN {X 0,Y 509.917,Z 177.783,A -85,B 0,C 180,E1 -5568.874,E2 -5568.874} C_VEL
LIN {X 0,Y 509.925,Z 177.78,A -85,B 0,C 180,E1 -5572.077,E2 -5572.077} C_VEL
LIN {X 0,Y 509.979,Z 177.772,A -85,B 0,C 180,E1 -5574.464,E2 -5574.464} C_VEL
LIN {X 0,Y 510.054,Z 177.766,A -85,B 0,C 180,E1 -5577.63,E2 -5577.63} C_VEL
LIN {X 0,Y 510.061,Z 177.765,A -85,B 0,C 180,E1 -5579.999,E2 -5579.999} C_VEL
LIN {X 0,Y 510.054,Z 177.763,A -85,B 0,C 180,E1 -5582.368,E2 -5582.368} C_VEL
LIN {X 0,Y 509.956,Z 177.776,A -85,B 0,C 180,E1 -5586.329,E2 -5586.329} C_VEL
LIN {X 0,Y 509.907,Z 177.782,A -85,B 0,C 180,E1 -5588.72,E2 -5588.72} C_VEL
LIN {X 0,Y 509.907,Z 177.783,A -85,B 0,C 180,E1 -5591.931,E2 -5591.931} C_VEL
LIN {X 0,Y 509.896,Z 177.785,A -85,B 0,C 180,E1 -5595.241,E2 -5595.241} C_VEL
LIN {X 0,Y 509.863,Z 177.788,A -85,B 0,C 180,E1 -5598.483,E2 -5598.483} C_VEL
LIN {X 0,Y 509.851,Z 177.789,A -85,B 0,C 180,E1 -5601.001,E2 -5601.001} C_VEL
LIN {X 0,Y 509.822,Z 177.793,A -85,B 0,C 180,E1 -5603.563,E2 -5603.563} C_VEL
LIN {X 0,Y 509.912,Z 177.782,A -85,B 0,C 180,E1 -5606.378,E2 -5606.378} C_VEL
LIN {X 0,Y 509.876,Z 177.786,A -85,B 0,C 180,E1 -5608.843,E2 -5608.843} C_VEL
LIN {X 0,Y 509.82,Z 177.792,A -85,B 0,C 180,E1 -5611.589,E2 -5611.589} C_VEL
LIN {X 0,Y 509.851,Z 177.791,A -85,B 0,C 180,E1 -5614.412,E2 -5614.412} C_VEL
LIN {X 0,Y 509.816,Z 177.795,A -85,B 0,C 180,E1 -5617.34,E2 -5617.34} C_VEL
LIN {X 0,Y 509.835,Z 177.791,A -85,B 0,C 180,E1 -5620.381,E2 -5620.381} C_VEL
LIN {X 0,Y 509.819,Z 177.792,A -85,B 0,C 180,E1 -5623.061,E2 -5623.061} C_VEL
LIN {X 0,Y 509.825,Z 177.793,A -85,B 0,C 180,E1 -5625.791,E2 -5625.791} C_VEL
LIN {X 0,Y 509.853,Z 177.791,A -85,B 0,C 180,E1 -5628.574,E2 -5628.574} C_VEL
LIN {X 0,Y 509.845,Z 177.79,A -85,B 0,C 180,E1 -5631.786,E2 -5631.786} C_VEL
LIN {X 0,Y 509.826,Z 177.793,A -85,B 0,C 180,E1 -5633.733,E2 -5633.733} C_VEL
LIN {X 0,Y 509.16,Z 177.875,A -85,B 0,C 180,E1 -5634.392,E2 -5634.392} C_VEL
LIN {X 0,Y 506.343,Z 178.227,A -85,B 0,C 180,E1 -5635.464,E2 -5635.464} C_VEL
LIN {X 0,Y 503.95,Z 178.526,A -85,B 0,C 180,E1 -5636.328,E2 -5636.328} C_VEL
LIN {X 0,Y 502.901,Z 178.654,A -85,B 0,C 180,E1 -5636.994,E2 -5636.994} C_VEL
LIN {X 0,Y 502.804,Z 178.665,A -85,B 0,C 180,E1 -5637.22,E2 -5637.22} C_VEL
LIN {X 0,Y 502.824,Z 178.667,A -85,B 0,C 180,E1 -5640.061,E2 -5640.061} C_VEL
LIN {X 0,Y 502.828,Z 178.665,A -85,B 0,C 180,E1 -5642.533,E2 -5642.533} C_VEL
LIN {X 0,Y 502.821,Z 178.667,A -85,B 0,C 180,E1 -5645.298,E2 -5645.298} C_VEL
LIN {X 0,Y 502.777,Z 178.672,A -85,B 0,C 180,E1 -5647.826,E2 -5647.826} C_VEL
LIN {X 0,Y 502.817,Z 178.666,A -85,B 0,C 180,E1 -5650.4,E2 -5650.4} C_VEL
LIN {X 0,Y 502.827,Z 178.666,A -85,B 0,C 180,E1 -5652.931,E2 -5652.931} C_VEL
LIN {X 0,Y 502.844,Z 178.665,A -85,B 0,C 180,E1 -5655.429,E2 -5655.429} C_VEL
LIN {X 0,Y 502.884,Z 178.657,A -85,B 0,C 180,E1 -5658.717,E2 -5658.717} C_VEL
LIN {X 0,Y 502.894,Z 178.657,A -85,B 0,C 180,E1 -5661.966,E2 -5661.966} C_VEL
LIN {X 0,Y 502.93,Z 178.652,A -85,B 0,C 180,E1 -5664.386,E2 -5664.386} C_VEL
LIN {X 0,Y 503.014,Z 178.64,A -85,B 0,C 180,E1 -5667.598,E2 -5667.598} C_VEL
LIN {X 0,Y 503.015,Z 178.641,A -85,B 0,C 180,E1 -5670,E2 -5670} C_VEL
LIN {X 0,Y 503.017,Z 178.642,A -85,B 0,C 180,E1 -5672.402,E2 -5672.402} C_VEL
LIN {X 0,Y 502.931,Z 178.651,A -85,B 0,C 180,E1 -5675.613,E2 -5675.613} C_VEL
LIN {X 0,Y 502.893,Z 178.655,A -85,B 0,C 180,E1 -5678.033,E2 -5678.033} C_VEL
LIN {X 0,Y 502.871,Z 178.659,A -85,B 0,C 180,E1 -5681.283,E2 -5681.283} C_VEL
LIN {X 0,Y 502.672,Z 178.685,A -85,B 0,C 180,E1 -5683.75,E2 -5683.75} C_VEL
LIN {X 0,Y 502.589,Z 178.771,A -85,B 0,C 180,E1 -5684.578,E2 -5684.578} C_VEL
LIN {X 0,Y 502.526,Z 184.031,A -85,B 0,C 180,E1 -5687.919,E2 -5687.919} C_VEL
LIN {X 0,Y 502.42,Z 189.482,A -85,B 0,C 180,E1 -5691.327,E2 -5691.327} C_VEL
LIN {X 0,Y 502.306,Z 193.718,A -85,B 0,C 180,E1 -5693.938,E2 -5693.938} C_VEL
LIN {X 0,Y 502.267,Z 198.067,A -85,B 0,C 180,E1 -5696.6,E2 -5696.6} C_VEL
LIN {X 0,Y 502.167,Z 203.371,A -85,B 0,C 180,E1 -5699.809,E2 -5699.809} C_VEL
LIN {X 0,Y 502.134,Z 208.512,A -85,B 0,C 180,E1 -5702.886,E2 -5702.886} C_VEL
LIN {X 0,Y 502.124,Z 211.571,A -85,B 0,C 180,E1 -5704.684,E2 -5704.684} C_VEL
LIN {X 0,Y 503.457,Z 220.926,A -85,B 0,C 180,E1 -5705.035,E2 -5705.035} C_VEL
LIN {X 0,Y 503.322,Z 230.185,A -85,B 0,C 180,E1 -5705.475,E2 -5705.475} C_VEL
LIN {X 0,Y 503.12,Z 239.35,A -85,B 0,C 180,E1 -5706.046,E2 -5706.046} C_VEL
LIN {X 0,Y 502.918,Z 248.721,A -85,B 0,C 180,E1 -5706.809,E2 -5706.809} C_VEL
LIN {X 0,Y 502.705,Z 255.811,A -85,B 0,C 180,E1 -5707.543,E2 -5707.543} C_VEL
LIN {X 0,Y 502.578,Z 261.18,A -85,B 0,C 180,E1 -5708.21,E2 -5708.21} C_VEL
LIN {X 0,Y 502.458,Z 266.514,A -85,B 0,C 180,E1 -5709.008,E2 -5709.008} C_VEL
LIN {X 0,Y 502.299,Z 272.139,A -85,B 0,C 180,E1 -5710.062,E2 -5710.062} C_VEL
LIN {X 0,Y 502.206,Z 276.51,A -85,B 0,C 180,E1 -5711.127,E2 -5711.127} C_VEL
LIN {X 0,Y 502.123,Z 279.744,A -85,B 0,C 180,E1 -5712.209,E2 -5712.209} C_VEL
LIN {X 0,Y 502.099,Z 281.847,A -85,B 0,C 180,E1 -5713.304,E2 -5713.304} C_VEL
LIN {X 0,Y 502.066,Z 282.943,A -85,B 0,C 180,E1 -5714.448,E2 -5714.448} C_VEL
LIN {X 0,Y 502.068,Z 282.98,A -85,B 0,C 180,E1 -5715.582,E2 -5715.582} C_VEL
LIN {X 0,Y 502.098,Z 281.98,A -85,B 0,C 180,E1 -5716.707,E2 -5716.707} C_VEL
LIN {X 0,Y 502.125,Z 279.791,A -85,B 0,C 180,E1 -5717.886,E2 -5717.886} C_VEL
LIN {X 0,Y 502.214,Z 276.134,A -85,B 0,C 180,E1 -5719.085,E2 -5719.085} C_VEL
LIN {X 0,Y 502.339,Z 270.926,A -85,B 0,C 180,E1 -5720.307,E2 -5720.307} C_VEL
LIN {X 0,Y 502.509,Z 265.318,A -85,B 0,C 180,E1 -5721.307,E2 -5721.307} C_VEL
LIN {X 0,Y 502.619,Z 258.54,A -85,B 0,C 180,E1 -5722.243,E2 -5722.243} C_VEL
LIN {X 0,Y 502.831,Z 251.151,A -85,B 0,C 180,E1 -5723.059,E2 -5723.059} C_VEL
LIN {X 0,Y 503.02,Z 244.047,A -85,B 0,C 180,E1 -5723.699,E2 -5723.699} C_VEL
LIN {X 0,Y 503.19,Z 235.352,A -85,B 0,C 180,E1 -5724.331,E2 -5724.331} C_VEL
LIN {X 0,Y 503.43,Z 224.83,A -85,B 0,C 180,E1 -5724.903,E2 -5724.903} C_VEL
LIN {X 0,Y 503.294,Z 218.631,A -85,B 0,C 180,E1 -5725.168,E2 -5725.168} C_VEL
LIN {X 0,Y 502.163,Z 211.835,A -85,B 0,C 180,E1 -5725.433,E2 -5725.433} C_VEL
LIN {X 0,Y 502.219,Z 206.213,A -85,B 0,C 180,E1 -5728.818,E2 -5728.818} C_VEL
LIN {X 0,Y 502.262,Z 201.267,A -85,B 0,C 180,E1 -5731.829,E2 -5731.829} C_VEL
LIN {X 0,Y 502.332,Z 197.277,A -85,B 0,C 180,E1 -5734.298,E2 -5734.298} C_VEL
LIN {X 0,Y 502.427,Z 192.268,A -85,B 0,C 180,E1 -5737.401,E2 -5737.401} C_VEL
LIN {X 0,Y 502.476,Z 187.533,A -85,B 0,C 180,E1 -5740.387,E2 -5740.387} C_VEL
LIN {X 0,Y 502.571,Z 183.51,A -85,B 0,C 180,E1 -5742.923,E2 -5742.923} C_VEL
LIN {X 0,Y 502.632,Z 179.63,A -85,B 0,C 180,E1 -5745.424,E2 -5745.424} C_VEL
LIN {X 0,Y 502.659,Z 178.689,A -85,B 0,C 180,E1 -5746.251,E2 -5746.251} C_VEL
LIN {X 0,Y 502.876,Z 178.662,A -85,B 0,C 180,E1 -5748.718,E2 -5748.718} C_VEL
LIN {X 0,Y 502.903,Z 178.658,A -85,B 0,C 180,E1 -5751.967,E2 -5751.967} C_VEL
LIN {X 0,Y 502.938,Z 178.656,A -85,B 0,C 180,E1 -5754.387,E2 -5754.387} C_VEL
LIN {X 0,Y 503.026,Z 178.641,A -85,B 0,C 180,E1 -5757.598,E2 -5757.598} C_VEL
LIN {X 0,Y 503.028,Z 178.64,A -85,B 0,C 180,E1 -5760.001,E2 -5760.001} C_VEL
LIN {X 0,Y 503.024,Z 178.642,A -85,B 0,C 180,E1 -5762.403,E2 -5762.403} C_VEL
LIN {X 0,Y 502.94,Z 178.651,A -85,B 0,C 180,E1 -5765.614,E2 -5765.614} C_VEL
LIN {X 0,Y 502.883,Z 178.659,A -85,B 0,C 180,E1 -5768.034,E2 -5768.034} C_VEL
LIN {X 0,Y 502.88,Z 178.658,A -85,B 0,C 180,E1 -5771.284,E2 -5771.284} C_VEL
LIN {X 0,Y 502.848,Z 178.661,A -85,B 0,C 180,E1 -5774.571,E2 -5774.571} C_VEL
LIN {X 0,Y 502.865,Z 178.66,A -85,B 0,C 180,E1 -5777.907,E2 -5777.907} C_VEL
LIN {X 0,Y 502.832,Z 178.664,A -85,B 0,C 180,E1 -5780.537,E2 -5780.537} C_VEL
LIN {X 0,Y 502.791,Z 178.671,A -85,B 0,C 180,E1 -5783.041,E2 -5783.041} C_VEL
LIN {X 0,Y 502.824,Z 178.665,A -85,B 0,C 180,E1 -5785.677,E2 -5785.677} C_VEL
LIN {X 0,Y 502.842,Z 178.663,A -85,B 0,C 180,E1 -5788.373,E2 -5788.373} C_VEL
LIN {X 0,Y 502.796,Z 178.668,A -85,B 0,C 180,E1 -5791.499,E2 -5791.499} C_VEL
LIN {X 0,Y 502.806,Z 178.666,A -85,B 0,C 180,E1 -5793.994,E2 -5793.994} C_VEL
LIN {X 0,Y 502.78,Z 178.671,A -85,B 0,C 180,E1 -5797.178,E2 -5797.178} C_VEL
LIN {X 0,Y 502.79,Z 178.67,A -85,B 0,C 180,E1 -5800.015,E2 -5800.015} C_VEL
LIN {X 0,Y 502.805,Z 178.669,A -85,B 0,C 180,E1 -5802.199,E2 -5802.199} C_VEL
LIN {X 0,Y 502.803,Z 178.669,A -85,B 0,C 180,E1 -5805.468,E2 -5805.468} C_VEL
LIN {X 0,Y 502.821,Z 178.666,A -85,B 0,C 180,E1 -5808.934,E2 -5808.934} C_VEL
LIN {X 0,Y 502.795,Z 178.671,A -85,B 0,C 180,E1 -5812.046,E2 -5812.046} C_VEL
LIN {X 0,Y 502.809,Z 178.674,A -85,B 0,C 180,E1 -5815.035,E2 -5815.035} C_VEL
LIN {X 0,Y 502.871,Z 178.737,A -85,B 0,C 180,E1 -5816.559,E2 -5816.559} C_VEL
LIN {X 0,Y 503.842,Z 184.88,A -85,B 0,C 180,E1 -5818.929,E2 -5818.929} C_VEL
LIN {X 0,Y 503.661,Z 191.276,A -85,B 0,C 180,E1 -5821.204,E2 -5821.204} C_VEL
LIN {X 0,Y 503.221,Z 200.573,A -85,B 0,C 180,E1 -5824.345,E2 -5824.345} C_VEL
LIN {X 0,Y 502.928,Z 209.511,A -85,B 0,C 180,E1 -5827.264,E2 -5827.264} C_VEL
LIN {X 0,Y 502.712,Z 218.027,A -85,B 0,C 180,E1 -5829.97,E2 -5829.97} C_VEL
LIN {X 0,Y 502.523,Z 227.597,A -85,B 0,C 180,E1 -5832.921,E2 -5832.921} C_VEL
LIN {X 0,Y 502.358,Z 237.227,A -85,B 0,C 180,E1 -5835.829,E2 -5835.829} C_VEL
LIN {X 0,Y 502.297,Z 247.038,A -85,B 0,C 180,E1 -5838.755,E2 -5838.755} C_VEL
LIN {X 0,Y 503.494,Z 259.355,A -85,B 0,C 180,E1 -5839.138,E2 -5839.138} C_VEL
LIN {X 0,Y 503.355,Z 268.675,A -85,B 0,C 180,E1 -5839.542,E2 -5839.542} C_VEL
LIN {X 0,Y 503.088,Z 279.069,A -85,B 0,C 180,E1 -5840.147,E2 -5840.147} C_VEL
LIN {X 0,Y 502.894,Z 287.26,A -85,B 0,C 180,E1 -5840.752,E2 -5840.752} C_VEL
LIN {X 0,Y 502.707,Z 295.042,A -85,B 0,C 180,E1 -5841.458,E2 -5841.458} C_VEL
LIN {X 0,Y 502.497,Z 303.194,A -85,B 0,C 180,E1 -5842.365,E2 -5842.365} C_VEL
LIN {X 0,Y 502.367,Z 310.214,A -85,B 0,C 180,E1 -5843.352,E2 -5843.352} C_VEL
LIN {X 0,Y 502.259,Z 315.97,A -85,B 0,C 180,E1 -5844.379,E2 -5844.379} C_VEL
LIN {X 0,Y 502.132,Z 321.208,A -85,B 0,C 180,E1 -5845.585,E2 -5845.585} C_VEL
LIN {X 0,Y 502.164,Z 323.894,A -85,B 0,C 180,E1 -5846.389,E2 -5846.389} C_VEL
LIN {X 0,Y 502.123,Z 326.837,A -85,B 0,C 180,E1 -5847.594,E2 -5847.594} C_VEL
LIN {X 0,Y 502.035,Z 328.106,A -85,B 0,C 180,E1 -5848.396,E2 -5848.396} C_VEL
LIN {X 0,Y 501.993,Z 328.898,A -85,B 0,C 180,E1 -5849.198,E2 -5849.198} C_VEL
LIN {X 0,Y 501.99,Z 329.203,A -85,B 0,C 180,E1 -5850,E2 -5850} C_VEL
LIN {X 0,Y 501.993,Z 328.911,A -85,B 0,C 180,E1 -5850.802,E2 -5850.802} C_VEL
LIN {X 0,Y 502.035,Z 328.128,A -85,B 0,C 180,E1 -5851.605,E2 -5851.605} C_VEL
LIN {X 0,Y 502.123,Z 326.868,A -85,B 0,C 180,E1 -5852.407,E2 -5852.407} C_VEL
LIN {X 0,Y 502.164,Z 323.946,A -85,B 0,C 180,E1 -5853.611,E2 -5853.611} C_VEL
LIN {X 0,Y 502.132,Z 321.271,A -85,B 0,C 180,E1 -5854.415,E2 -5854.415} C_VEL
LIN {X 0,Y 502.26,Z 316.053,A -85,B 0,C 180,E1 -5855.621,E2 -5855.621} C_VEL
LIN {X 0,Y 502.4,Z 309.15,A -85,B 0,C 180,E1 -5856.829,E2 -5856.829} C_VEL
LIN {X 0,Y 502.546,Z 301.609,A -85,B 0,C 180,E1 -5857.837,E2 -5857.837} C_VEL
LIN {X 0,Y 502.715,Z 295.197,A -85,B 0,C 180,E1 -5858.542,E2 -5858.542} C_VEL
LIN {X 0,Y 502.894,Z 287.432,A -85,B 0,C 180,E1 -5859.249,E2 -5859.249} C_VEL
LIN {X 0,Y 503.097,Z 279.261,A -85,B 0,C 180,E1 -5859.853,E2 -5859.853} C_VEL
LIN {X 0,Y 503.326,Z 268.894,A -85,B 0,C 180,E1 -5860.459,E2 -5860.459} C_VEL
LIN {X 0,Y 503.418,Z 258.166,A -85,B 0,C 180,E1 -5860.914,E2 -5860.914} C_VEL
LIN {X 0,Y 502.297,Z 247.287,A -85,B 0,C 180,E1 -5861.245,E2 -5861.245} C_VEL
LIN {X 0,Y 502.403,Z 236.14,A -85,B 0,C 180,E1 -5864.584,E2 -5864.584} C_VEL
LIN {X 0,Y 502.598,Z 226.575,A -85,B 0,C 180,E1 -5867.496,E2 -5867.496} C_VEL
LIN {X 0,Y 502.826,Z 215.663,A -85,B 0,C 180,E1 -5870.88,E2 -5870.88} C_VEL
LIN {X 0,Y 503.074,Z 206.154,A -85,B 0,C 180,E1 -5873.9,E2 -5873.9} C_VEL
LIN {X 0,Y 503.382,Z 197.636,A -85,B 0,C 180,E1 -5876.678,E2 -5876.678} C_VEL
LIN {X 0,Y 503.761,Z 188.699,A -85,B 0,C 180,E1 -5879.681,E2 -5879.681} C_VEL
LIN {X 0,Y 503.801,Z 184.683,A -85,B 0,C 180,E1 -5881.075,E2 -5881.075} C_VEL
LIN {X 0,Y 502.84,Z 178.665,A -85,B 0,C 180,E1 -5883.33,E2 -5883.33} C_VEL
LIN {X 0,Y 502.776,Z 178.67,A -85,B 0,C 180,E1 -5885.951,E2 -5885.951} C_VEL
LIN {X 0,Y 502.804,Z 178.669,A -85,B 0,C 180,E1 -5888.976,E2 -5888.976} C_VEL
LIN {X 0,Y 502.798,Z 178.668,A -85,B 0,C 180,E1 -5892.139,E2 -5892.139} C_VEL
LIN {X 0,Y 502.789,Z 178.67,A -85,B 0,C 180,E1 -5895.47,E2 -5895.47} C_VEL
LIN {X 0,Y 502.798,Z 178.668,A -85,B 0,C 180,E1 -5897.861,E2 -5897.861} C_VEL
LIN {X 0,Y 502.804,Z 178.666,A -85,B 0,C 180,E1 -5901.024,E2 -5901.024} C_VEL
LIN {X 0,Y 502.779,Z 178.671,A -85,B 0,C 180,E1 -5904.169,E2 -5904.169} C_VEL
LIN {X 0,Y 502.837,Z 178.664,A -85,B 0,C 180,E1 -5906.993,E2 -5906.993} C_VEL
LIN {X 0,Y 502.819,Z 178.665,A -85,B 0,C 180,E1 -5910.065,E2 -5910.065} C_VEL
LIN {X 0,Y 502.832,Z 178.663,A -85,B 0,C 180,E1 -5912.533,E2 -5912.533} C_VEL
LIN {X 0,Y 502.808,Z 178.666,A -85,B 0,C 180,E1 -5915.305,E2 -5915.305} C_VEL
LIN {X 0,Y 502.785,Z 178.67,A -85,B 0,C 180,E1 -5917.826,E2 -5917.826} C_VEL
LIN {X 0,Y 502.828,Z 178.663,A -85,B 0,C 180,E1 -5920.4,E2 -5920.4} C_VEL
LIN {X 0,Y 502.823,Z 178.664,A -85,B 0,C 180,E1 -5922.931,E2 -5922.931} C_VEL
LIN {X 0,Y 502.85,Z 178.662,A -85,B 0,C 180,E1 -5925.429,E2 -5925.429} C_VEL
LIN {X 0,Y 502.881,Z 178.659,A -85,B 0,C 180,E1 -5928.716,E2 -5928.716} C_VEL
LIN {X 0,Y 502.885,Z 178.657,A -85,B 0,C 180,E1 -5931.966,E2 -5931.966} C_VEL
LIN {X 0,Y 502.934,Z 178.649,A -85,B 0,C 180,E1 -5934.386,E2 -5934.386} C_VEL
LIN {X 0,Y 503.024,Z 178.642,A -85,B 0,C 180,E1 -5937.597,E2 -5937.597} C_VEL
LIN {X 0,Y 503.032,Z 178.64,A -85,B 0,C 180,E1 -5939.999,E2 -5939.999} C_VEL
LIN {X 0,Y 503.025,Z 178.638,A -85,B 0,C 180,E1 -5942.402,E2 -5942.402} C_VEL
LIN {X 0,Y 502.933,Z 178.65,A -85,B 0,C 180,E1 -5945.613,E2 -5945.613} C_VEL
LIN {X 0,Y 502.883,Z 178.658,A -85,B 0,C 180,E1 -5948.033,E2 -5948.033} C_VEL
LIN {X 0,Y 502.88,Z 178.658,A -85,B 0,C 180,E1 -5951.282,E2 -5951.282} C_VEL
LIN {X 0,Y 502.847,Z 178.663,A -85,B 0,C 180,E1 -5954.57,E2 -5954.57} C_VEL
LIN {X 0,Y 502.824,Z 178.665,A -85,B 0,C 180,E1 -5957.907,E2 -5957.907} C_VEL
LIN {X 0,Y 502.83,Z 178.666,A -85,B 0,C 180,E1 -5960.535,E2 -5960.535} C_VEL
LIN {X 0,Y 502.788,Z 178.671,A -85,B 0,C 180,E1 -5963.04,E2 -5963.04} C_VEL
LIN {X 0,Y 502.822,Z 178.666,A -85,B 0,C 180,E1 -5965.676,E2 -5965.676} C_VEL
LIN {X 0,Y 502.84,Z 178.665,A -85,B 0,C 180,E1 -5968.372,E2 -5968.372} C_VEL
LIN {X 0,Y 502.792,Z 178.667,A -85,B 0,C 180,E1 -5971.498,E2 -5971.498} C_VEL
LIN {X 0,Y 502.803,Z 178.669,A -85,B 0,C 180,E1 -5974.443,E2 -5974.443} C_VEL
LIN {X 0,Y 502.778,Z 178.671,A -85,B 0,C 180,E1 -5977.177,E2 -5977.177} C_VEL
LIN {X 0,Y 502.784,Z 178.671,A -85,B 0,C 180,E1 -5980.014,E2 -5980.014} C_VEL
LIN {X 0,Y 502.799,Z 178.67,A -85,B 0,C 180,E1 -5982.198,E2 -5982.198} C_VEL
LIN {X 0,Y 502.796,Z 178.668,A -85,B 0,C 180,E1 -5985.467,E2 -5985.467} C_VEL
LIN {X 0,Y 502.815,Z 178.666,A -85,B 0,C 180,E1 -5988.933,E2 -5988.933} C_VEL
LIN {X 0,Y 502.788,Z 178.669,A -85,B 0,C 180,E1 -5992.045,E2 -5992.045} C_VEL
LIN {X 0,Y 502.805,Z 178.668,A -85,B 0,C 180,E1 -5995.034,E2 -5995.034} C_VEL
LIN {X 0,Y 502.804,Z 178.665,A -85,B 0,C 180,E1 -5997.22,E2 -5997.22} C_VEL
LIN {X 0,Y 502.106,Z 178.755,A -85,B 0,C 180,E1 -5997.888,E2 -5997.888} C_VEL
LIN {X 0,Y 499.248,Z 179.111,A -85,B 0,C 180,E1 -5998.974,E2 -5998.974} C_VEL
LIN {X 0,Y 496.856,Z 179.409,A -85,B 0,C 180,E1 -5999.849,E2 -5999.849} C_VEL
LIN {X 0,Y 495.838,Z 179.535,A -85,B 0,C 180,E1 -6000.525,E2 -6000.525} C_VEL
LIN {X 0,Y 495.758,Z 179.543,A -85,B 0,C 180,E1 -6000.754,E2 -6000.754} C_VEL
LIN {X 0,Y 495.784,Z 179.544,A -85,B 0,C 180,E1 -6003.931,E2 -6003.931} C_VEL
LIN {X 0,Y 495.758,Z 179.545,A -85,B 0,C 180,E1 -6007.137,E2 -6007.137} C_VEL
LIN {X 0,Y 495.77,Z 179.544,A -85,B 0,C 180,E1 -6010.109,E2 -6010.109} C_VEL
LIN {X 0,Y 495.779,Z 179.542,A -85,B 0,C 180,E1 -6012.681,E2 -6012.681} C_VEL
LIN {X 0,Y 495.786,Z 179.542,A -85,B 0,C 180,E1 -6015.217,E2 -6015.217} C_VEL
LIN {X 0,Y 495.865,Z 179.532,A -85,B 0,C 180,E1 -6018.555,E2 -6018.555} C_VEL
LIN {X 0,Y 495.865,Z 179.532,A -85,B 0,C 180,E1 -6021.852,E2 -6021.852} C_VEL
LIN {X 0,Y 495.888,Z 179.529,A -85,B 0,C 180,E1 -6024.306,E2 -6024.306} C_VEL
LIN {X 0,Y 495.983,Z 179.515,A -85,B 0,C 180,E1 -6027.563,E2 -6027.563} C_VEL
LIN {X 0,Y 495.986,Z 179.516,A -85,B 0,C 180,E1 -6030,E2 -6030} C_VEL
LIN {X 0,Y 495.986,Z 179.518,A -85,B 0,C 180,E1 -6032.436,E2 -6032.436} C_VEL
LIN {X 0,Y 495.888,Z 179.528,A -85,B 0,C 180,E1 -6035.693,E2 -6035.693} C_VEL
LIN {X 0,Y 495.864,Z 179.531,A -85,B 0,C 180,E1 -6038.148,E2 -6038.148} C_VEL
LIN {X 0,Y 495.839,Z 179.534,A -85,B 0,C 180,E1 -6041.445,E2 -6041.445} C_VEL
LIN {X 0,Y 495.595,Z 179.568,A -85,B 0,C 180,E1 -6043.95,E2 -6043.95} C_VEL
LIN {X 0,Y 495.542,Z 179.89,A -85,B 0,C 180,E1 -6044.79,E2 -6044.79} C_VEL
LIN {X 0,Y 495.435,Z 185.079,A -85,B 0,C 180,E1 -6048.12,E2 -6048.12} C_VEL
LIN {X 0,Y 495.366,Z 189.281,A -85,B 0,C 180,E1 -6050.774,E2 -6050.774} C_VEL
LIN {X 0,Y 495.255,Z 193.515,A -85,B 0,C 180,E1 -6053.412,E2 -6053.412} C_VEL
LIN {X 0,Y 495.216,Z 197.864,A -85,B 0,C 180,E1 -6056.1,E2 -6056.1} C_VEL
LIN {X 0,Y 495.106,Z 202.389,A -85,B 0,C 180,E1 -6058.857,E2 -6058.857} C_VEL
LIN {X 0,Y 495.075,Z 207.064,A -85,B 0,C 180,E1 -6061.685,E2 -6061.685} C_VEL
LIN {X 0,Y 495.056,Z 211.941,A -85,B 0,C 180,E1 -6064.535,E2 -6064.535} C_VEL
LIN {X 0,Y 496.476,Z 221.451,A -85,B 0,C 180,E1 -6064.902,E2 -6064.902} C_VEL
LIN {X 0,Y 496.365,Z 229.782,A -85,B 0,C 180,E1 -6065.3,E2 -6065.3} C_VEL
LIN {X 0,Y 496.132,Z 238.612,A -85,B 0,C 180,E1 -6065.847,E2 -6065.847} C_VEL
LIN {X 0,Y 495.944,Z 247.218,A -85,B 0,C 180,E1 -6066.525,E2 -6066.525} C_VEL
LIN {X 0,Y 495.673,Z 256.144,A -85,B 0,C 180,E1 -6067.44,E2 -6067.44} C_VEL
LIN {X 0,Y 495.483,Z 263.18,A -85,B 0,C 180,E1 -6068.357,E2 -6068.357} C_VEL
LIN {X 0,Y 495.376,Z 268.25,A -85,B 0,C 180,E1 -6069.171,E2 -6069.171} C_VEL
LIN {X 0,Y 495.182,Z 274.062,A -85,B 0,C 180,E1 -6070.339,E2 -6070.339} C_VEL
LIN {X 0,Y 495.116,Z 277.329,A -85,B 0,C 180,E1 -6071.21,E2 -6071.21} C_VEL
LIN {X 0,Y 495.037,Z 280.588,A -85,B 0,C 180,E1 -6072.42,E2 -6072.42} C_VEL
LIN {X 0,Y 495.006,Z 282.563,A -85,B 0,C 180,E1 -6073.609,E2 -6073.609} C_VEL
LIN {X 0,Y 494.972,Z 283.404,A -85,B 0,C 180,E1 -6074.772,E2 -6074.772} C_VEL
LIN {X 0,Y 494.985,Z 283.181,A -85,B 0,C 180,E1 -6075.917,E2 -6075.917} C_VEL
LIN {X 0,Y 495.009,Z 281.888,A -85,B 0,C 180,E1 -6077.041,E2 -6077.041} C_VEL
LIN {X 0,Y 495.063,Z 279.522,A -85,B 0,C 180,E1 -6078.149,E2 -6078.149} C_VEL
LIN {X 0,Y 495.137,Z 276.111,A -85,B 0,C 180,E1 -6079.239,E2 -6079.239} C_VEL
LIN {X 0,Y 495.261,Z 271.571,A -85,B 0,C 180,E1 -6080.316,E2 -6080.316} C_VEL
LIN {X 0,Y 495.449,Z 265.746,A -85,B 0,C 180,E1 -6081.382,E2 -6081.382} C_VEL
LIN {X 0,Y 495.62,Z 258.178,A -85,B 0,C 180,E1 -6082.43,E2 -6082.43} C_VEL
LIN {X 0,Y 495.816,Z 251.12,A -85,B 0,C 180,E1 -6083.212,E2 -6083.212} C_VEL
LIN {X 0,Y 496.067,Z 243.119,A -85,B 0,C 180,E1 -6083.929,E2 -6083.929} C_VEL
LIN {X 0,Y 496.273,Z 233.021,A -85,B 0,C 180,E1 -6084.631,E2 -6084.631} C_VEL
LIN {X 0,Y 496.506,Z 223.96,A -85,B 0,C 180,E1 -6085.097,E2 -6085.097} C_VEL
LIN {X 0,Y 496.067,Z 217.945,A -85,B 0,C 180,E1 -6085.358,E2 -6085.358} C_VEL
LIN {X 0,Y 495.102,Z 212.123,A -85,B 0,C 180,E1 -6085.588,E2 -6085.588} C_VEL
LIN {X 0,Y 495.098,Z 207.497,A -85,B 0,C 180,E1 -6088.398,E2 -6088.398} C_VEL
LIN {X 0,Y 495.175,Z 202.226,A -85,B 0,C 180,E1 -6091.638,E2 -6091.638} C_VEL
LIN {X 0,Y 495.263,Z 198.595,A -85,B 0,C 180,E1 -6093.903,E2 -6093.903} C_VEL
LIN {X 0,Y 495.294,Z 194.294,A -85,B 0,C 180,E1 -6096.591,E2 -6096.591} C_VEL
LIN {X 0,Y 495.418,Z 189.807,A -85,B 0,C 180,E1 -6099.435,E2 -6099.435} C_VEL
LIN {X 0,Y 495.509,Z 184.725,A -85,B 0,C 180,E1 -6102.672,E2 -6102.672} C_VEL
LIN {X 0,Y 495.591,Z 180.844,A -85,B 0,C 180,E1 -6105.212,E2 -6105.212} C_VEL
LIN {X 0,Y 495.573,Z 179.571,A -85,B 0,C 180,E1 -6106.05,E2 -6106.05} C_VEL
LIN {X 0,Y 495.846,Z 179.538,A -85,B 0,C 180,E1 -6108.556,E2 -6108.556} C_VEL
LIN {X 0,Y 495.874,Z 179.533,A -85,B 0,C 180,E1 -6111.853,E2 -6111.853} C_VEL
LIN {X 0,Y 495.896,Z 179.533,A -85,B 0,C 180,E1 -6114.307,E2 -6114.307} C_VEL
LIN {X 0,Y 495.994,Z 179.517,A -85,B 0,C 180,E1 -6117.564,E2 -6117.564} C_VEL
LIN {X 0,Y 496,Z 179.516,A -85,B 0,C 180,E1 -6120.001,E2 -6120.001} C_VEL
LIN {X 0,Y 495.993,Z 179.518,A -85,B 0,C 180,E1 -6122.437,E2 -6122.437} C_VEL
LIN {X 0,Y 495.898,Z 179.529,A -85,B 0,C 180,E1 -6125.694,E2 -6125.694} C_VEL
LIN {X 0,Y 495.839,Z 179.537,A -85,B 0,C 180,E1 -6128.149,E2 -6128.149} C_VEL
LIN {X 0,Y 495.854,Z 179.534,A -85,B 0,C 180,E1 -6131.446,E2 -6131.446} C_VEL
LIN {X 0,Y 495.793,Z 179.541,A -85,B 0,C 180,E1 -6134.783,E2 -6134.783} C_VEL
LIN {X 0,Y 495.788,Z 179.544,A -85,B 0,C 180,E1 -6137.319,E2 -6137.319} C_VEL
LIN {X 0,Y 495.781,Z 179.543,A -85,B 0,C 180,E1 -6139.89,E2 -6139.89} C_VEL
LIN {X 0,Y 495.761,Z 179.545,A -85,B 0,C 180,E1 -6142.861,E2 -6142.861} C_VEL
LIN {X 0,Y 495.783,Z 179.541,A -85,B 0,C 180,E1 -6146.069,E2 -6146.069} C_VEL
LIN {X 0,Y 495.774,Z 179.545,A -85,B 0,C 180,E1 -6148.815,E2 -6148.815} C_VEL
LIN {X 0,Y 495.759,Z 179.544,A -85,B 0,C 180,E1 -6151.726,E2 -6151.726} C_VEL
LIN {X 0,Y 495.771,Z 179.545,A -85,B 0,C 180,E1 -6154.694,E2 -6154.694} C_VEL
LIN {X 0,Y 495.731,Z 179.548,A -85,B 0,C 180,E1 -6157.562,E2 -6157.562} C_VEL
LIN {X 0,Y 495.768,Z 179.545,A -85,B 0,C 180,E1 -6160.7,E2 -6160.7} C_VEL
LIN {X 0,Y 495.736,Z 179.55,A -85,B 0,C 180,E1 -6164.001,E2 -6164.001} C_VEL
LIN {X 0,Y 495.727,Z 179.552,A -85,B 0,C 180,E1 -6167.117,E2 -6167.117} C_VEL
LIN {X 0,Y 495.76,Z 179.545,A -85,B 0,C 180,E1 -6169.953,E2 -6169.953} C_VEL
LIN {X 0,Y 495.732,Z 179.55,A -85,B 0,C 180,E1 -6172.553,E2 -6172.553} C_VEL
LIN {X 0,Y 495.785,Z 179.549,A -85,B 0,C 180,E1 -6175.457,E2 -6175.457} C_VEL
LIN {X 0,Y 495.813,Z 179.584,A -85,B 0,C 180,E1 -6176.318,E2 -6176.318} C_VEL
LIN {X 0,Y 496.883,Z 186.189,A -85,B 0,C 180,E1 -6178.918,E2 -6178.918} C_VEL
LIN {X 0,Y 496.622,Z 192.872,A -85,B 0,C 180,E1 -6181.331,E2 -6181.331} C_VEL
LIN {X 0,Y 496.184,Z 201.79,A -85,B 0,C 180,E1 -6184.405,E2 -6184.405} C_VEL
LIN {X 0,Y 495.858,Z 211.112,A -85,B 0,C 180,E1 -6187.5,E2 -6187.5} C_VEL
LIN {X 0,Y 495.63,Z 220.58,A -85,B 0,C 180,E1 -6190.535,E2 -6190.535} C_VEL
LIN {X 0,Y 495.422,Z 228.734,A -85,B 0,C 180,E1 -6193.094,E2 -6193.094} C_VEL
LIN {X 0,Y 495.258,Z 238.338,A -85,B 0,C 180,E1 -6196.04,E2 -6196.04} C_VEL
LIN {X 0,Y 495.23,Z 246.75,A -85,B 0,C 180,E1 -6198.592,E2 -6198.592} C_VEL
LIN {X 0,Y 496.501,Z 260.147,A -85,B 0,C 180,E1 -6199.035,E2 -6199.035} C_VEL
LIN {X 0,Y 496.309,Z 270.132,A -85,B 0,C 180,E1 -6199.495,E2 -6199.495} C_VEL
LIN {X 0,Y 496.087,Z 278.669,A -85,B 0,C 180,E1 -6200.006,E2 -6200.006} C_VEL
LIN {X 0,Y 495.922,Z 285.638,A -85,B 0,C 180,E1 -6200.518,E2 -6200.518} C_VEL
LIN {X 0,Y 495.686,Z 293.638,A -85,B 0,C 180,E1 -6201.233,E2 -6201.233} C_VEL
LIN {X 0,Y 495.451,Z 301.108,A -85,B 0,C 180,E1 -6202.05,E2 -6202.05} C_VEL
LIN {X 0,Y 495.29,Z 308.964,A -85,B 0,C 180,E1 -6203.114,E2 -6203.114} C_VEL
LIN {X 0,Y 495.189,Z 315.625,A -85,B 0,C 180,E1 -6204.299,E2 -6204.299} C_VEL
LIN {X 0,Y 495.037,Z 320.868,A -85,B 0,C 180,E1 -6205.522,E2 -6205.522} C_VEL
LIN {X 0,Y 495.084,Z 323.56,A -85,B 0,C 180,E1 -6206.338,E2 -6206.338} C_VEL
LIN {X 0,Y 495.027,Z 326.506,A -85,B 0,C 180,E1 -6207.559,E2 -6207.559} C_VEL
LIN {X 0,Y 494.962,Z 327.78,A -85,B 0,C 180,E1 -6208.373,E2 -6208.373} C_VEL
LIN {X 0,Y 494.913,Z 328.573,A -85,B 0,C 180,E1 -6209.186,E2 -6209.186} C_VEL
LIN {X 0,Y 494.907,Z 328.878,A -85,B 0,C 180,E1 -6210,E2 -6210} C_VEL
LIN {X 0,Y 494.913,Z 328.588,A -85,B 0,C 180,E1 -6210.814,E2 -6210.814} C_VEL
LIN {X 0,Y 494.962,Z 327.806,A -85,B 0,C 180,E1 -6211.627,E2 -6211.627} C_VEL
LIN {X 0,Y 495.027,Z 326.544,A -85,B 0,C 180,E1 -6212.441,E2 -6212.441} C_VEL
LIN {X 0,Y 495.084,Z 323.621,A -85,B 0,C 180,E1 -6213.663,E2 -6213.663} C_VEL
LIN {X 0,Y 495.037,Z 320.942,A -85,B 0,C 180,E1 -6214.479,E2 -6214.479} C_VEL
LIN {X 0,Y 495.189,Z 315.723,A -85,B 0,C 180,E1 -6215.702,E2 -6215.702} C_VEL
LIN {X 0,Y 495.333,Z 308.808,A -85,B 0,C 180,E1 -6216.927,E2 -6216.927} C_VEL
LIN {X 0,Y 495.471,Z 301.261,A -85,B 0,C 180,E1 -6217.95,E2 -6217.95} C_VEL
LIN {X 0,Y 495.664,Z 294.841,A -85,B 0,C 180,E1 -6218.665,E2 -6218.665} C_VEL
LIN {X 0,Y 495.886,Z 287.067,A -85,B 0,C 180,E1 -6219.38,E2 -6219.38} C_VEL
LIN {X 0,Y 496.048,Z 280.382,A -85,B 0,C 180,E1 -6219.892,E2 -6219.892} C_VEL
LIN {X 0,Y 496.251,Z 272.233,A -85,B 0,C 180,E1 -6220.403,E2 -6220.403} C_VEL
LIN {X 0,Y 496.446,Z 264.016,A -85,B 0,C 180,E1 -6220.811,E2 -6220.811} C_VEL
LIN {X 0,Y 496.288,Z 257.663,A -85,B 0,C 180,E1 -6221.073,E2 -6221.073} C_VEL
LIN {X 0,Y 495.231,Z 247.015,A -85,B 0,C 180,E1 -6221.408,E2 -6221.408} C_VEL
LIN {X 0,Y 495.333,Z 235.935,A -85,B 0,C 180,E1 -6224.797,E2 -6224.797} C_VEL
LIN {X 0,Y 495.573,Z 225.064,A -85,B 0,C 180,E1 -6228.164,E2 -6228.164} C_VEL
LIN {X 0,Y 495.843,Z 214.14,A -85,B 0,C 180,E1 -6231.625,E2 -6231.625} C_VEL
LIN {X 0,Y 496.226,Z 203.334,A -85,B 0,C 180,E1 -6235.144,E2 -6235.144} C_VEL
LIN {X 0,Y 496.58,Z 194.076,A -85,B 0,C 180,E1 -6238.257,E2 -6238.257} C_VEL
LIN {X 0,Y 496.875,Z 187.264,A -85,B 0,C 180,E1 -6240.611,E2 -6240.611} C_VEL
LIN {X 0,Y 496.556,Z 183.795,A -85,B 0,C 180,E1 -6241.874,E2 -6241.874} C_VEL
LIN {X 0,Y 495.795,Z 179.542,A -85,B 0,C 180,E1 -6243.514,E2 -6243.514} C_VEL
LIN {X 0,Y 495.731,Z 179.551,A -85,B 0,C 180,E1 -6246.544,E2 -6246.544} C_VEL
LIN {X 0,Y 495.76,Z 179.543,A -85,B 0,C 180,E1 -6249.638,E2 -6249.638} C_VEL
LIN {X 0,Y 495.741,Z 179.547,A -85,B 0,C 180,E1 -6252.507,E2 -6252.507} C_VEL
LIN {X 0,Y 495.741,Z 179.547,A -85,B 0,C 180,E1 -6255.141,E2 -6255.141} C_VEL
LIN {X 0,Y 495.754,Z 179.547,A -85,B 0,C 180,E1 -6258.218,E2 -6258.218} C_VEL
LIN {X 0,Y 495.753,Z 179.544,A -85,B 0,C 180,E1 -6261.408,E2 -6261.408} C_VEL
LIN {X 0,Y 495.752,Z 179.547,A -85,B 0,C 180,E1 -6264.462,E2 -6264.462} C_VEL
LIN {X 0,Y 495.772,Z 179.543,A -85,B 0,C 180,E1 -6267.406,E2 -6267.406} C_VEL
LIN {X 0,Y 495.77,Z 179.543,A -85,B 0,C 180,E1 -6270.253,E2 -6270.253} C_VEL
LIN {X 0,Y 495.828,Z 179.536,A -85,B 0,C 180,E1 -6273.251,E2 -6273.251} C_VEL
LIN {X 0,Y 495.747,Z 179.545,A -85,B 0,C 180,E1 -6276.612,E2 -6276.612} C_VEL
LIN {X 0,Y 495.783,Z 179.541,A -85,B 0,C 180,E1 -6279.324,E2 -6279.324} C_VEL
LIN {X 0,Y 495.786,Z 179.542,A -85,B 0,C 180,E1 -6281.828,E2 -6281.828} C_VEL
LIN {X 0,Y 495.829,Z 179.536,A -85,B 0,C 180,E1 -6284.548,E2 -6284.548} C_VEL
LIN {X 0,Y 495.833,Z 179.535,A -85,B 0,C 180,E1 -6287.965,E2 -6287.965} C_VEL
LIN {X 0,Y 495.838,Z 179.535,A -85,B 0,C 180,E1 -6291.03,E2 -6291.03} C_VEL
LIN {X 0,Y 495.863,Z 179.533,A -85,B 0,C 180,E1 -6293.489,E2 -6293.489} C_VEL
LIN {X 0,Y 495.842,Z 179.535,A -85,B 0,C 180,E1 -6296.749,E2 -6296.749} C_VEL
LIN {X 0,Y 495.871,Z 179.529,A -85,B 0,C 180,E1 -6298.375,E2 -6298.375} C_VEL
LIN {X 0,Y 495.966,Z 179.519,A -85,B 0,C 180,E1 -6300.811,E2 -6300.811} C_VEL
LIN {X 0,Y 495.994,Z 179.514,A -85,B 0,C 180,E1 -6302.436,E2 -6302.436} C_VEL
LIN {X 0,Y 495.89,Z 179.527,A -85,B 0,C 180,E1 -6305.693,E2 -6305.693} C_VEL
LIN {X 0,Y 495.839,Z 179.536,A -85,B 0,C 180,E1 -6308.148,E2 -6308.148} C_VEL
LIN {X 0,Y 495.854,Z 179.534,A -85,B 0,C 180,E1 -6311.444,E2 -6311.444} C_VEL
LIN {X 0,Y 495.792,Z 179.541,A -85,B 0,C 180,E1 -6314.782,E2 -6314.782} C_VEL
LIN {X 0,Y 495.765,Z 179.543,A -85,B 0,C 180,E1 -6317.318,E2 -6317.318} C_VEL
LIN {X 0,Y 495.772,Z 179.542,A -85,B 0,C 180,E1 -6319.889,E2 -6319.889} C_VEL
LIN {X 0,Y 495.759,Z 179.546,A -85,B 0,C 180,E1 -6322.859,E2 -6322.859} C_VEL
LIN {X 0,Y 495.781,Z 179.543,A -85,B 0,C 180,E1 -6326.067,E2 -6326.067} C_VEL
LIN {X 0,Y 495.771,Z 179.543,A -85,B 0,C 180,E1 -6328.814,E2 -6328.814} C_VEL
LIN {X 0,Y 495.755,Z 179.544,A -85,B 0,C 180,E1 -6331.724,E2 -6331.724} C_VEL
LIN {X 0,Y 495.773,Z 179.544,A -85,B 0,C 180,E1 -6334.694,E2 -6334.694} C_VEL
LIN {X 0,Y 495.728,Z 179.549,A -85,B 0,C 180,E1 -6337.56,E2 -6337.56} C_VEL
LIN {X 0,Y 495.763,Z 179.545,A -85,B 0,C 180,E1 -6340.699,E2 -6340.699} C_VEL
LIN {X 0,Y 495.73,Z 179.549,A -85,B 0,C 180,E1 -6344,E2 -6344} C_VEL
LIN {X 0,Y 495.72,Z 179.549,A -85,B 0,C 180,E1 -6347.116,E2 -6347.116} C_VEL
LIN {X 0,Y 495.753,Z 179.548,A -85,B 0,C 180,E1 -6349.952,E2 -6349.952} C_VEL
LIN {X 0,Y 495.725,Z 179.55,A -85,B 0,C 180,E1 -6352.552,E2 -6352.552} C_VEL
LIN {X 0,Y 495.78,Z 179.543,A -85,B 0,C 180,E1 -6355.457,E2 -6355.457} C_VEL
LIN {X 0,Y 495.753,Z 179.544,A -85,B 0,C 180,E1 -6358.363,E2 -6358.363} C_VEL
LIN {X 0,Y 495.758,Z 179.543,A -85,B 0,C 180,E1 -6360.754,E2 -6360.754} C_VEL
LIN {X 0,Y 495.096,Z 179.63,A -85,B 0,C 180,E1 -6361.433,E2 -6361.433} C_VEL
LIN {X 0,Y 492.235,Z 179.984,A -85,B 0,C 180,E1 -6362.535,E2 -6362.535} C_VEL
LIN {X 0,Y 489.824,Z 180.284,A -85,B 0,C 180,E1 -6363.424,E2 -6363.424} C_VEL
LIN {X 0,Y 488.808,Z 180.411,A -85,B 0,C 180,E1 -6364.11,E2 -6364.11} C_VEL
LIN {X 0,Y 488.735,Z 180.418,A -85,B 0,C 180,E1 -6364.342,E2 -6364.342} C_VEL
LIN {X 0,Y 488.72,Z 180.422,A -85,B 0,C 180,E1 -6367.153,E2 -6367.153} C_VEL
LIN {X 0,Y 488.721,Z 180.421,A -85,B 0,C 180,E1 -6369.81,E2 -6369.81} C_VEL
LIN {X 0,Y 488.726,Z 180.419,A -85,B 0,C 180,E1 -6372.423,E2 -6372.423} C_VEL
LIN {X 0,Y 488.756,Z 180.417,A -85,B 0,C 180,E1 -6374.999,E2 -6374.999} C_VEL
LIN {X 0,Y 488.823,Z 180.41,A -85,B 0,C 180,E1 -6378.388,E2 -6378.388} C_VEL
LIN {X 0,Y 488.81,Z 180.411,A -85,B 0,C 180,E1 -6381.733,E2 -6381.733} C_VEL
LIN {X 0,Y 488.847,Z 180.405,A -85,B 0,C 180,E1 -6384.224,E2 -6384.224} C_VEL
LIN {X 0,Y 488.95,Z 180.391,A -85,B 0,C 180,E1 -6387.528,E2 -6387.528} C_VEL
LIN {X 0,Y 488.958,Z 180.392,A -85,B 0,C 180,E1 -6390,E2 -6390} C_VEL
LIN {X 0,Y 488.953,Z 180.393,A -85,B 0,C 180,E1 -6392.471,E2 -6392.471} C_VEL
LIN {X 0,Y 488.848,Z 180.405,A -85,B 0,C 180,E1 -6395.776,E2 -6395.776} C_VEL
LIN {X 0,Y 488.809,Z 180.411,A -85,B 0,C 180,E1 -6398.266,E2 -6398.266} C_VEL
LIN {X 0,Y 488.791,Z 180.412,A -85,B 0,C 180,E1 -6401.613,E2 -6401.613} C_VEL
LIN {X 0,Y 488.49,Z 180.523,A -85,B 0,C 180,E1 -6404.689,E2 -6404.689} C_VEL
LIN {X 0,Y 488.373,Z 186.013,A -85,B 0,C 180,E1 -6408.239,E2 -6408.239} C_VEL
LIN {X 0,Y 488.285,Z 190.49,A -85,B 0,C 180,E1 -6411.09,E2 -6411.09} C_VEL
LIN {X 0,Y 488.181,Z 194.761,A -85,B 0,C 180,E1 -6413.772,E2 -6413.772} C_VEL
LIN {X 0,Y 488.161,Z 199.144,A -85,B 0,C 180,E1 -6416.507,E2 -6416.507} C_VEL
LIN {X 0,Y 488.018,Z 203.714,A -85,B 0,C 180,E1 -6419.317,E2 -6419.317} C_VEL
LIN {X 0,Y 487.98,Z 208.45,A -85,B 0,C 180,E1 -6422.2,E2 -6422.2} C_VEL
LIN {X 0,Y 487.961,Z 212.075,A -85,B 0,C 180,E1 -6424.373,E2 -6424.373} C_VEL
LIN {X 0,Y 489.448,Z 221.488,A -85,B 0,C 180,E1 -6424.743,E2 -6424.743} C_VEL
LIN {X 0,Y 489.395,Z 230.097,A -85,B 0,C 180,E1 -6425.161,E2 -6425.161} C_VEL
LIN {X 0,Y 489.15,Z 238.307,A -85,B 0,C 180,E1 -6425.672,E2 -6425.672} C_VEL
LIN {X 0,Y 488.933,Z 247.443,A -85,B 0,C 180,E1 -6426.396,E2 -6426.396} C_VEL
LIN {X 0,Y 488.663,Z 256.134,A -85,B 0,C 180,E1 -6427.293,E2 -6427.293} C_VEL
LIN {X 0,Y 488.456,Z 263.213,A -85,B 0,C 180,E1 -6428.221,E2 -6428.221} C_VEL
LIN {X 0,Y 488.327,Z 268.071,A -85,B 0,C 180,E1 -6429,E2 -6429} C_VEL
LIN {X 0,Y 488.142,Z 273.242,A -85,B 0,C 180,E1 -6430.022,E2 -6430.022} C_VEL
LIN {X 0,Y 488.055,Z 276.848,A -85,B 0,C 180,E1 -6430.935,E2 -6430.935} C_VEL
LIN {X 0,Y 487.966,Z 280.174,A -85,B 0,C 180,E1 -6432.045,E2 -6432.045} C_VEL
LIN {X 0,Y 487.952,Z 281.596,A -85,B 0,C 180,E1 -6432.732,E2 -6432.732} C_VEL
LIN {X 0,Y 487.906,Z 283.289,A -85,B 0,C 180,E1 -6433.929,E2 -6433.929} C_VEL
LIN {X 0,Y 487.887,Z 283.809,A -85,B 0,C 180,E1 -6435.104,E2 -6435.104} C_VEL
LIN {X 0,Y 487.923,Z 283.204,A -85,B 0,C 180,E1 -6436.261,E2 -6436.261} C_VEL
LIN {X 0,Y 487.931,Z 281.596,A -85,B 0,C 180,E1 -6437.394,E2 -6437.394} C_VEL
LIN {X 0,Y 488.017,Z 278.967,A -85,B 0,C 180,E1 -6438.514,E2 -6438.514} C_VEL
LIN {X 0,Y 488.121,Z 274.843,A -85,B 0,C 180,E1 -6439.738,E2 -6439.738} C_VEL
LIN {X 0,Y 488.271,Z 270.42,A -85,B 0,C 180,E1 -6440.706,E2 -6440.706} C_VEL
LIN {X 0,Y 488.436,Z 264.063,A -85,B 0,C 180,E1 -6441.779,E2 -6441.779} C_VEL
LIN {X 0,Y 488.622,Z 258.242,A -85,B 0,C 180,E1 -6442.572,E2 -6442.572} C_VEL
LIN {X 0,Y 488.821,Z 251.118,A -85,B 0,C 180,E1 -6443.367,E2 -6443.367} C_VEL
LIN {X 0,Y 489.145,Z 242.229,A -85,B 0,C 180,E1 -6444.164,E2 -6444.164} C_VEL
LIN {X 0,Y 489.316,Z 232.727,A -85,B 0,C 180,E1 -6444.81,E2 -6444.81} C_VEL
LIN {X 0,Y 489.576,Z 223.199,A -85,B 0,C 180,E1 -6445.295,E2 -6445.295} C_VEL
LIN {X 0,Y 488.541,Z 215.551,A -85,B 0,C 180,E1 -6445.615,E2 -6445.615} C_VEL
LIN {X 0,Y 488.02,Z 212.413,A -85,B 0,C 180,E1 -6445.746,E2 -6445.746} C_VEL
LIN {X 0,Y 488.024,Z 207.497,A -85,B 0,C 180,E1 -6448.774,E2 -6448.774} C_VEL
LIN {X 0,Y 488.114,Z 202.889,A -85,B 0,C 180,E1 -6451.632,E2 -6451.632} C_VEL
LIN {X 0,Y 488.195,Z 198.457,A -85,B 0,C 180,E1 -6454.414,E2 -6454.414} C_VEL
LIN {X 0,Y 488.296,Z 194.19,A -85,B 0,C 180,E1 -6457.133,E2 -6457.133} C_VEL
LIN {X 0,Y 488.359,Z 190.027,A -85,B 0,C 180,E1 -6459.796,E2 -6459.796} C_VEL
LIN {X 0,Y 488.468,Z 185.984,A -85,B 0,C 180,E1 -6462.414,E2 -6462.414} C_VEL
LIN {X 0,Y 488.557,Z 182.055,A -85,B 0,C 180,E1 -6464.994,E2 -6464.994} C_VEL
LIN {X 0,Y 488.523,Z 180.779,A -85,B 0,C 180,E1 -6465.845,E2 -6465.845} C_VEL
LIN {X 0,Y 488.723,Z 180.427,A -85,B 0,C 180,E1 -6467.544,E2 -6467.544} C_VEL
LIN {X 0,Y 488.766,Z 180.418,A -85,B 0,C 180,E1 -6470.065,E2 -6470.065} C_VEL
LIN {X 0,Y 488.872,Z 180.406,A -85,B 0,C 180,E1 -6472.721,E2 -6472.721} C_VEL
LIN {X 0,Y 488.81,Z 180.414,A -85,B 0,C 180,E1 -6475.052,E2 -6475.052} C_VEL
LIN {X 0,Y 488.962,Z 180.393,A -85,B 0,C 180,E1 -6477.529,E2 -6477.529} C_VEL
LIN {X 0,Y 488.957,Z 180.392,A -85,B 0,C 180,E1 -6480.824,E2 -6480.824} C_VEL
LIN {X 0,Y 488.961,Z 180.394,A -85,B 0,C 180,E1 -6482.472,E2 -6482.472} C_VEL
LIN {X 0,Y 488.857,Z 180.406,A -85,B 0,C 180,E1 -6485.776,E2 -6485.776} C_VEL
LIN {X 0,Y 488.788,Z 180.416,A -85,B 0,C 180,E1 -6488.267,E2 -6488.267} C_VEL
LIN {X 0,Y 488.808,Z 180.413,A -85,B 0,C 180,E1 -6491.613,E2 -6491.613} C_VEL
LIN {X 0,Y 488.765,Z 180.418,A -85,B 0,C 180,E1 -6495.001,E2 -6495.001} C_VEL
LIN {X 0,Y 488.758,Z 180.419,A -85,B 0,C 180,E1 -6498.443,E2 -6498.443} C_VEL
LIN {X 0,Y 488.709,Z 180.424,A -85,B 0,C 180,E1 -6501.071,E2 -6501.071} C_VEL
LIN {X 0,Y 488.682,Z 180.426,A -85,B 0,C 180,E1 -6503.747,E2 -6503.747} C_VEL
LIN {X 0,Y 488.794,Z 180.413,A -85,B 0,C 180,E1 -6506.944,E2 -6506.944} C_VEL
LIN {X 0,Y 488.712,Z 180.423,A -85,B 0,C 180,E1 -6510.363,E2 -6510.363} C_VEL
LIN {X 0,Y 488.737,Z 180.421,A -85,B 0,C 180,E1 -6513.484,E2 -6513.484} C_VEL
LIN {X 0,Y 488.684,Z 180.426,A -85,B 0,C 180,E1 -6516.355,E2 -6516.355} C_VEL
LIN {X 0,Y 488.703,Z 180.426,A -85,B 0,C 180,E1 -6519.255,E2 -6519.255} C_VEL
LIN {X 0,Y 488.709,Z 180.426,A -85,B 0,C 180,E1 -6521.6,E2 -6521.6} C_VEL
LIN {X 0,Y 488.714,Z 180.426,A -85,B 0,C 180,E1 -6524.802,E2 -6524.802} C_VEL
LIN {X 0,Y 488.693,Z 180.427,A -85,B 0,C 180,E1 -6527.475,E2 -6527.475} C_VEL
LIN {X 0,Y 488.735,Z 180.422,A -85,B 0,C 180,E1 -6529.677,E2 -6529.677} C_VEL
LIN {X 0,Y 488.684,Z 180.43,A -85,B 0,C 180,E1 -6532.842,E2 -6532.842} C_VEL
LIN {X 0,Y 488.788,Z 180.59,A -85,B 0,C 180,E1 -6536.145,E2 -6536.145} C_VEL
LIN {X 0,Y 489.743,Z 186.202,A -85,B 0,C 180,E1 -6538.413,E2 -6538.413} C_VEL
LIN {X 0,Y 489.826,Z 190.021,A -85,B 0,C 180,E1 -6539.856,E2 -6539.856} C_VEL
LIN {X 0,Y 489.369,Z 198.574,A -85,B 0,C 180,E1 -6542.924,E2 -6542.924} C_VEL
LIN {X 0,Y 488.939,Z 208.319,A -85,B 0,C 180,E1 -6546.267,E2 -6546.267} C_VEL
LIN {X 0,Y 488.68,Z 217.156,A -85,B 0,C 180,E1 -6549.197,E2 -6549.197} C_VEL
LIN {X 0,Y 488.438,Z 227.167,A -85,B 0,C 180,E1 -6552.413,E2 -6552.413} C_VEL
LIN {X 0,Y 488.228,Z 236.698,A -85,B 0,C 180,E1 -6555.409,E2 -6555.409} C_VEL
LIN {X 0,Y 488.153,Z 246.461,A -85,B 0,C 180,E1 -6558.425,E2 -6558.425} C_VEL
LIN {X 0,Y 489.439,Z 259.717,A -85,B 0,C 180,E1 -6558.875,E2 -6558.875} C_VEL
LIN {X 0,Y 489.306,Z 269.722,A -85,B 0,C 180,E1 -6559.343,E2 -6559.343} C_VEL
LIN {X 0,Y 489.065,Z 278.274,A -85,B 0,C 180,E1 -6559.861,E2 -6559.861} C_VEL
LIN {X 0,Y 488.845,Z 286.492,A -85,B 0,C 180,E1 -6560.484,E2 -6560.484} C_VEL
LIN {X 0,Y 488.645,Z 293.268,A -85,B 0,C 180,E1 -6561.106,E2 -6561.106} C_VEL
LIN {X 0,Y 488.464,Z 299.03,A -85,B 0,C 180,E1 -6561.728,E2 -6561.728} C_VEL
LIN {X 0,Y 488.3,Z 305.469,A -85,B 0,C 180,E1 -6562.557,E2 -6562.557} C_VEL
LIN {X 0,Y 488.181,Z 310.82,A -85,B 0,C 180,E1 -6563.387,E2 -6563.387} C_VEL
LIN {X 0,Y 488.093,Z 315.283,A -85,B 0,C 180,E1 -6564.215,E2 -6564.215} C_VEL
LIN {X 0,Y 487.949,Z 320.531,A -85,B 0,C 180,E1 -6565.457,E2 -6565.457} C_VEL
LIN {X 0,Y 488.004,Z 323.228,A -85,B 0,C 180,E1 -6566.284,E2 -6566.284} C_VEL
LIN {X 0,Y 487.935,Z 326.176,A -85,B 0,C 180,E1 -6567.524,E2 -6567.524} C_VEL
LIN {X 0,Y 487.891,Z 327.453,A -85,B 0,C 180,E1 -6568.349,E2 -6568.349} C_VEL
LIN {X 0,Y 487.836,Z 328.249,A -85,B 0,C 180,E1 -6569.175,E2 -6569.175} C_VEL
LIN {X 0,Y 487.827,Z 328.554,A -85,B 0,C 180,E1 -6570,E2 -6570} C_VEL
LIN {X 0,Y 487.836,Z 328.265,A -85,B 0,C 180,E1 -6570.826,E2 -6570.826} C_VEL
LIN {X 0,Y 487.891,Z 327.482,A -85,B 0,C 180,E1 -6571.651,E2 -6571.651} C_VEL
LIN {X 0,Y 487.935,Z 326.218,A -85,B 0,C 180,E1 -6572.477,E2 -6572.477} C_VEL
LIN {X 0,Y 488.005,Z 323.294,A -85,B 0,C 180,E1 -6573.716,E2 -6573.716} C_VEL
LIN {X 0,Y 487.949,Z 320.612,A -85,B 0,C 180,E1 -6574.544,E2 -6574.544} C_VEL
LIN {X 0,Y 488.094,Z 315.386,A -85,B 0,C 180,E1 -6575.785,E2 -6575.785} C_VEL
LIN {X 0,Y 488.275,Z 308.458,A -85,B 0,C 180,E1 -6577.028,E2 -6577.028} C_VEL
LIN {X 0,Y 488.417,Z 300.903,A -85,B 0,C 180,E1 -6578.065,E2 -6578.065} C_VEL
LIN {X 0,Y 488.621,Z 294.471,A -85,B 0,C 180,E1 -6578.791,E2 -6578.791} C_VEL
LIN {X 0,Y 488.807,Z 287.914,A -85,B 0,C 180,E1 -6579.413,E2 -6579.413} C_VEL
LIN {X 0,Y 489.045,Z 279.979,A -85,B 0,C 180,E1 -6580.035,E2 -6580.035} C_VEL
LIN {X 0,Y 489.253,Z 271.804,A -85,B 0,C 180,E1 -6580.554,E2 -6580.554} C_VEL
LIN {X 0,Y 489.476,Z 263.551,A -85,B 0,C 180,E1 -6580.967,E2 -6580.967} C_VEL
LIN {X 0,Y 489.105,Z 256.295,A -85,B 0,C 180,E1 -6581.264,E2 -6581.264} C_VEL
LIN {X 0,Y 488.154,Z 246.763,A -85,B 0,C 180,E1 -6581.576,E2 -6581.576} C_VEL
LIN {X 0,Y 488.327,Z 234.58,A -85,B 0,C 180,E1 -6585.363,E2 -6585.363} C_VEL
LIN {X 0,Y 488.506,Z 224.807,A -85,B 0,C 180,E1 -6588.452,E2 -6588.452} C_VEL
LIN {X 0,Y 488.778,Z 215.328,A -85,B 0,C 180,E1 -6591.51,E2 -6591.51} C_VEL
LIN {X 0,Y 489.201,Z 204.286,A -85,B 0,C 180,E1 -6595.166,E2 -6595.166} C_VEL
LIN {X 0,Y 489.584,Z 195.171,A -85,B 0,C 180,E1 -6598.276,E2 -6598.276} C_VEL
LIN {X 0,Y 489.902,Z 188.565,A -85,B 0,C 180,E1 -6600.599,E2 -6600.599} C_VEL
LIN {X 0,Y 489.467,Z 184.507,A -85,B 0,C 180,E1 -6602.097,E2 -6602.097} C_VEL
LIN {X 0,Y 488.737,Z 180.422,A -85,B 0,C 180,E1 -6603.677,E2 -6603.677} C_VEL
LIN {X 0,Y 488.685,Z 180.428,A -85,B 0,C 180,E1 -6606.355,E2 -6606.355} C_VEL
LIN {X 0,Y 488.704,Z 180.427,A -85,B 0,C 180,E1 -6609.254,E2 -6609.254} C_VEL
LIN {X 0,Y 488.71,Z 180.423,A -85,B 0,C 180,E1 -6611.6,E2 -6611.6} C_VEL
LIN {X 0,Y 488.705,Z 180.423,A -85,B 0,C 180,E1 -6614.803,E2 -6614.803} C_VEL
LIN {X 0,Y 488.692,Z 180.423,A -85,B 0,C 180,E1 -6617.474,E2 -6617.474} C_VEL
LIN {X 0,Y 488.704,Z 180.424,A -85,B 0,C 180,E1 -6620.746,E2 -6620.746} C_VEL
LIN {X 0,Y 488.681,Z 180.426,A -85,B 0,C 180,E1 -6623.868,E2 -6623.868} C_VEL
LIN {X 0,Y 488.743,Z 180.419,A -85,B 0,C 180,E1 -6626.877,E2 -6626.877} C_VEL
LIN {X 0,Y 488.728,Z 180.422,A -85,B 0,C 180,E1 -6629.781,E2 -6629.781} C_VEL
LIN {X 0,Y 488.796,Z 180.411,A -85,B 0,C 180,E1 -6633.056,E2 -6633.056} C_VEL
LIN {X 0,Y 488.684,Z 180.426,A -85,B 0,C 180,E1 -6636.254,E2 -6636.254} C_VEL
LIN {X 0,Y 488.751,Z 180.417,A -85,B 0,C 180,E1 -6639.175,E2 -6639.175} C_VEL
LIN {X 0,Y 488.754,Z 180.418,A -85,B 0,C 180,E1 -6641.631,E2 -6641.631} C_VEL
LIN {X 0,Y 488.767,Z 180.417,A -85,B 0,C 180,E1 -6644.999,E2 -6644.999} C_VEL
LIN {X 0,Y 488.81,Z 180.411,A -85,B 0,C 180,E1 -6648.387,E2 -6648.387} C_VEL
LIN {X 0,Y 488.789,Z 180.413,A -85,B 0,C 180,E1 -6651.733,E2 -6651.733} C_VEL
LIN {X 0,Y 488.849,Z 180.404,A -85,B 0,C 180,E1 -6654.224,E2 -6654.224} C_VEL
LIN {X 0,Y 488.962,Z 180.394,A -85,B 0,C 180,E1 -6657.528,E2 -6657.528} C_VEL
LIN {X 0,Y 488.974,Z 180.391,A -85,B 0,C 180,E1 -6659.999,E2 -6659.999} C_VEL
LIN {X 0,Y 488.962,Z 180.39,A -85,B 0,C 180,E1 -6662.471,E2 -6662.471} C_VEL
LIN {X 0,Y 488.848,Z 180.404,A -85,B 0,C 180,E1 -6665.775,E2 -6665.775} C_VEL
LIN {X 0,Y 488.788,Z 180.413,A -85,B 0,C 180,E1 -6668.266,E2 -6668.266} C_VEL
LIN {X 0,Y 488.808,Z 180.411,A -85,B 0,C 180,E1 -6671.612,E2 -6671.612} C_VEL
LIN {X 0,Y 488.764,Z 180.416,A -85,B 0,C 180,E1 -6674.999,E2 -6674.999} C_VEL
LIN {X 0,Y 488.748,Z 180.419,A -85,B 0,C 180,E1 -6678.441,E2 -6678.441} C_VEL
LIN {X 0,Y 488.708,Z 180.423,A -85,B 0,C 180,E1 -6681.07,E2 -6681.07} C_VEL
LIN {X 0,Y 488.679,Z 180.426,A -85,B 0,C 180,E1 -6683.745,E2 -6683.745} C_VEL
LIN {X 0,Y 488.792,Z 180.414,A -85,B 0,C 180,E1 -6686.943,E2 -6686.943} C_VEL
LIN {X 0,Y 488.708,Z 180.423,A -85,B 0,C 180,E1 -6690.362,E2 -6690.362} C_VEL
LIN {X 0,Y 488.734,Z 180.421,A -85,B 0,C 180,E1 -6693.483,E2 -6693.483} C_VEL
LIN {X 0,Y 488.686,Z 180.426,A -85,B 0,C 180,E1 -6696.355,E2 -6696.355} C_VEL
LIN {X 0,Y 488.697,Z 180.422,A -85,B 0,C 180,E1 -6699.253,E2 -6699.253} C_VEL
LIN {X 0,Y 488.704,Z 180.424,A -85,B 0,C 180,E1 -6701.599,E2 -6701.599} C_VEL
LIN {X 0,Y 488.707,Z 180.424,A -85,B 0,C 180,E1 -6704.8,E2 -6704.8} C_VEL
LIN {X 0,Y 488.686,Z 180.427,A -85,B 0,C 180,E1 -6707.474,E2 -6707.474} C_VEL
LIN {X 0,Y 488.727,Z 180.421,A -85,B 0,C 180,E1 -6709.676,E2 -6709.676} C_VEL
LIN {X 0,Y 488.677,Z 180.427,A -85,B 0,C 180,E1 -6712.841,E2 -6712.841} C_VEL
LIN {X 0,Y 488.73,Z 180.421,A -85,B 0,C 180,E1 -6715.887,E2 -6715.887} C_VEL
LIN {X 0,Y 488.69,Z 180.425,A -85,B 0,C 180,E1 -6718.82,E2 -6718.82} C_VEL
LIN {X 0,Y 488.74,Z 180.42,A -85,B 0,C 180,E1 -6721.671,E2 -6721.671} C_VEL
LIN {X 0,Y 488.735,Z 180.418,A -85,B 0,C 180,E1 -6724.342,E2 -6724.342} C_VEL
LIN {X 0,Y 488.091,Z 180.502,A -85,B 0,C 180,E1 -6725.03,E2 -6725.03} C_VEL
LIN {X 0,Y 485.225,Z 180.863,A -85,B 0,C 180,E1 -6726.146,E2 -6726.146} C_VEL
LIN {X 0,Y 482.779,Z 181.166,A -85,B 0,C 180,E1 -6727.046,E2 -6727.046} C_VEL
LIN {X 0,Y 481.721,Z 181.295,A -85,B 0,C 180,E1 -6727.742,E2 -6727.742} C_VEL
LIN {X 0,Y 481.631,Z 181.304,A -85,B 0,C 180,E1 -6727.977,E2 -6727.977} C_VEL
LIN {X 0,Y 481.7,Z 181.296,A -85,B 0,C 180,E1 -6730.393,E2 -6730.393} C_VEL
LIN {X 0,Y 481.683,Z 181.301,A -85,B 0,C 180,E1 -6733.033,E2 -6733.033} C_VEL
LIN {X 0,Y 481.688,Z 181.298,A -85,B 0,C 180,E1 -6735.638,E2 -6735.638} C_VEL
LIN {X 0,Y 481.786,Z 181.286,A -85,B 0,C 180,E1 -6738.216,E2 -6738.216} C_VEL
LIN {X 0,Y 481.755,Z 181.29,A -85,B 0,C 180,E1 -6741.611,E2 -6741.611} C_VEL
LIN {X 0,Y 481.808,Z 181.281,A -85,B 0,C 180,E1 -6744.139,E2 -6744.139} C_VEL
LIN {X 0,Y 481.917,Z 181.267,A -85,B 0,C 180,E1 -6747.492,E2 -6747.492} C_VEL
LIN {X 0,Y 481.929,Z 181.267,A -85,B 0,C 180,E1 -6750,E2 -6750} C_VEL
LIN {X 0,Y 481.92,Z 181.269,A -85,B 0,C 180,E1 -6752.507,E2 -6752.507} C_VEL
LIN {X 0,Y 481.808,Z 181.282,A -85,B 0,C 180,E1 -6755.86,E2 -6755.86} C_VEL
LIN {X 0,Y 481.755,Z 181.291,A -85,B 0,C 180,E1 -6758.388,E2 -6758.388} C_VEL
LIN {X 0,Y 481.736,Z 181.29,A -85,B 0,C 180,E1 -6761.785,E2 -6761.785} C_VEL
LIN {X 0,Y 481.437,Z 181.494,A -85,B 0,C 180,E1 -6764.801,E2 -6764.801} C_VEL
LIN {X 0,Y 481.324,Z 186.176,A -85,B 0,C 180,E1 -6767.856,E2 -6767.856} C_VEL
LIN {X 0,Y 481.244,Z 190.778,A -85,B 0,C 180,E1 -6770.833,E2 -6770.833} C_VEL
LIN {X 0,Y 481.12,Z 196.008,A -85,B 0,C 180,E1 -6774.143,E2 -6774.143} C_VEL
LIN {X 0,Y 481.043,Z 200.526,A -85,B 0,C 180,E1 -6776.978,E2 -6776.978} C_VEL
LIN {X 0,Y 480.923,Z 205.089,A -85,B 0,C 180,E1 -6779.792,E2 -6779.792} C_VEL
LIN {X 0,Y 480.901,Z 209.87,A -85,B 0,C 180,E1 -6782.733,E2 -6782.733} C_VEL
LIN {X 0,Y 480.891,Z 212.298,A -85,B 0,C 180,E1 -6784.208,E2 -6784.208} C_VEL
LIN {X 0,Y 482.48,Z 222.307,A -85,B 0,C 180,E1 -6784.617,E2 -6784.617} C_VEL
LIN {X 0,Y 482.41,Z 230.293,A -85,B 0,C 180,E1 -6785.013,E2 -6785.013} C_VEL
LIN {X 0,Y 482.15,Z 238.95,A -85,B 0,C 180,E1 -6785.562,E2 -6785.562} C_VEL
LIN {X 0,Y 481.929,Z 248.19,A -85,B 0,C 180,E1 -6786.312,E2 -6786.312} C_VEL
LIN {X 0,Y 481.602,Z 257.168,A -85,B 0,C 180,E1 -6787.273,E2 -6787.273} C_VEL
LIN {X 0,Y 481.418,Z 263.721,A -85,B 0,C 180,E1 -6788.154,E2 -6788.154} C_VEL
LIN {X 0,Y 481.213,Z 270.435,A -85,B 0,C 180,E1 -6789.283,E2 -6789.283} C_VEL
LIN {X 0,Y 481.02,Z 276.008,A -85,B 0,C 180,E1 -6790.56,E2 -6790.56} C_VEL
LIN {X 0,Y 480.959,Z 278.004,A -85,B 0,C 180,E1 -6791.114,E2 -6791.114} C_VEL
LIN {X 0,Y 480.866,Z 281.03,A -85,B 0,C 180,E1 -6792.245,E2 -6792.245} C_VEL
LIN {X 0,Y 480.842,Z 282.997,A -85,B 0,C 180,E1 -6793.389,E2 -6793.389} C_VEL
LIN {X 0,Y 480.798,Z 283.969,A -85,B 0,C 180,E1 -6794.558,E2 -6794.558} C_VEL
LIN {X 0,Y 480.804,Z 283.911,A -85,B 0,C 180,E1 -6795.745,E2 -6795.745} C_VEL
LIN {X 0,Y 480.844,Z 282.771,A -85,B 0,C 180,E1 -6796.953,E2 -6796.953} C_VEL
LIN {X 0,Y 480.889,Z 280.335,A -85,B 0,C 180,E1 -6798.189,E2 -6798.189} C_VEL
LIN {X 0,Y 480.96,Z 278.426,A -85,B 0,C 180,E1 -6798.887,E2 -6798.887} C_VEL
LIN {X 0,Y 481.094,Z 274.373,A -85,B 0,C 180,E1 -6800.003,E2 -6800.003} C_VEL
LIN {X 0,Y 481.282,Z 269.031,A -85,B 0,C 180,E1 -6801.105,E2 -6801.105} C_VEL
LIN {X 0,Y 481.435,Z 263.421,A -85,B 0,C 180,E1 -6802.026,E2 -6802.026} C_VEL
LIN {X 0,Y 481.681,Z 256.063,A -85,B 0,C 180,E1 -6802.998,E2 -6802.998} C_VEL
LIN {X 0,Y 481.95,Z 246.883,A -85,B 0,C 180,E1 -6803.932,E2 -6803.932} C_VEL
LIN {X 0,Y 482.192,Z 239.143,A -85,B 0,C 180,E1 -6804.553,E2 -6804.553} C_VEL
LIN {X 0,Y 482.408,Z 230.894,A -85,B 0,C 180,E1 -6805.082,E2 -6805.082} C_VEL
LIN {X 0,Y 482.536,Z 222.161,A -85,B 0,C 180,E1 -6805.515,E2 -6805.515} C_VEL
LIN {X 0,Y 480.953,Z 212.687,A -85,B 0,C 180,E1 -6805.924,E2 -6805.924} C_VEL
LIN {X 0,Y 480.955,Z 207.361,A -85,B 0,C 180,E1 -6809.241,E2 -6809.241} C_VEL
LIN {X 0,Y 481.06,Z 202.757,A -85,B 0,C 180,E1 -6812.129,E2 -6812.129} C_VEL
LIN {X 0,Y 481.159,Z 198.365,A -85,B 0,C 180,E1 -6814.94,E2 -6814.94} C_VEL
LIN {X 0,Y 481.225,Z 194.085,A -85,B 0,C 180,E1 -6817.685,E2 -6817.685} C_VEL
LIN {X 0,Y 481.324,Z 189.948,A -85,B 0,C 180,E1 -6820.378,E2 -6820.378} C_VEL
LIN {X 0,Y 481.423,Z 185.917,A -85,B 0,C 180,E1 -6823.025,E2 -6823.025} C_VEL
LIN {X 0,Y 481.48,Z 182.013,A -85,B 0,C 180,E1 -6825.633,E2 -6825.633} C_VEL
LIN {X 0,Y 481.54,Z 181.322,A -85,B 0,C 180,E1 -6826.497,E2 -6826.497} C_VEL
LIN {X 0,Y 481.744,Z 181.294,A -85,B 0,C 180,E1 -6828.216,E2 -6828.216} C_VEL
LIN {X 0,Y 481.764,Z 181.291,A -85,B 0,C 180,E1 -6831.613,E2 -6831.613} C_VEL
LIN {X 0,Y 481.817,Z 181.286,A -85,B 0,C 180,E1 -6834.14,E2 -6834.14} C_VEL
LIN {X 0,Y 481.929,Z 181.269,A -85,B 0,C 180,E1 -6837.493,E2 -6837.493} C_VEL
LIN {X 0,Y 481.908,Z 181.27,A -85,B 0,C 180,E1 -6840.836,E2 -6840.836} C_VEL
LIN {X 0,Y 481.928,Z 181.27,A -85,B 0,C 180,E1 -6842.508,E2 -6842.508} C_VEL
LIN {X 0,Y 481.818,Z 181.284,A -85,B 0,C 180,E1 -6845.861,E2 -6845.861} C_VEL
LIN {X 0,Y 481.743,Z 181.292,A -85,B 0,C 180,E1 -6848.389,E2 -6848.389} C_VEL
LIN {X 0,Y 481.753,Z 181.291,A -85,B 0,C 180,E1 -6851.785,E2 -6851.785} C_VEL
LIN {X 0,Y 481.745,Z 181.292,A -85,B 0,C 180,E1 -6855.225,E2 -6855.225} C_VEL
LIN {X 0,Y 481.715,Z 181.295,A -85,B 0,C 180,E1 -6858.722,E2 -6858.722} C_VEL
LIN {X 0,Y 481.648,Z 181.303,A -85,B 0,C 180,E1 -6861.395,E2 -6861.395} C_VEL
LIN {X 0,Y 481.664,Z 181.302,A -85,B 0,C 180,E1 -6864.114,E2 -6864.114} C_VEL
LIN {X 0,Y 481.749,Z 181.29,A -85,B 0,C 180,E1 -6867.139,E2 -6867.139} C_VEL
LIN {X 0,Y 481.681,Z 181.299,A -85,B 0,C 180,E1 -6869.741,E2 -6869.741} C_VEL
LIN {X 0,Y 481.675,Z 181.299,A -85,B 0,C 180,E1 -6872.674,E2 -6872.674} C_VEL
LIN {X 0,Y 481.639,Z 181.306,A -85,B 0,C 180,E1 -6875.71,E2 -6875.71} C_VEL
LIN {X 0,Y 481.673,Z 181.3,A -85,B 0,C 180,E1 -6878.859,E2 -6878.859} C_VEL
LIN {X 0,Y 481.654,Z 181.304,A -85,B 0,C 180,E1 -6881.913,E2 -6881.913} C_VEL
LIN {X 0,Y 481.662,Z 181.303,A -85,B 0,C 180,E1 -6884.458,E2 -6884.458} C_VEL
LIN {X 0,Y 481.649,Z 181.304,A -85,B 0,C 180,E1 -6887.84,E2 -6887.84} C_VEL
LIN {X 0,Y 481.682,Z 181.301,A -85,B 0,C 180,E1 -6890.651,E2 -6890.651} C_VEL
LIN {X 0,Y 481.632,Z 181.309,A -85,B 0,C 180,E1 -6893.376,E2 -6893.376} C_VEL
LIN {X 0,Y 481.751,Z 181.427,A -85,B 0,C 180,E1 -6895.892,E2 -6895.892} C_VEL
LIN {X 0,Y 482.787,Z 187.512,A -85,B 0,C 180,E1 -6898.395,E2 -6898.395} C_VEL
LIN {X 0,Y 482.826,Z 191.295,A -85,B 0,C 180,E1 -6899.856,E2 -6899.856} C_VEL
LIN {X 0,Y 482.398,Z 199.116,A -85,B 0,C 180,E1 -6902.711,E2 -6902.711} C_VEL
LIN {X 0,Y 481.953,Z 208.207,A -85,B 0,C 180,E1 -6905.902,E2 -6905.902} C_VEL
LIN {X 0,Y 481.642,Z 217.497,A -85,B 0,C 180,E1 -6909.047,E2 -6909.047} C_VEL
LIN {X 0,Y 481.387,Z 226.952,A -85,B 0,C 180,E1 -6912.146,E2 -6912.146} C_VEL
LIN {X 0,Y 481.157,Z 236.463,A -85,B 0,C 180,E1 -6915.19,E2 -6915.19} C_VEL
LIN {X 0,Y 481.07,Z 246.223,A -85,B 0,C 180,E1 -6918.268,E2 -6918.268} C_VEL
LIN {X 0,Y 482.349,Z 259.486,A -85,B 0,C 180,E1 -6918.716,E2 -6918.716} C_VEL
LIN {X 0,Y 482.312,Z 269.358,A -85,B 0,C 180,E1 -6919.187,E2 -6919.187} C_VEL
LIN {X 0,Y 482.06,Z 277.917,A -85,B 0,C 180,E1 -6919.712,E2 -6919.712} C_VEL
LIN {X 0,Y 481.835,Z 286.137,A -85,B 0,C 180,E1 -6920.344,E2 -6920.344} C_VEL
LIN {X 0,Y 481.588,Z 293.944,A -85,B 0,C 180,E1 -6921.08,E2 -6921.08} C_VEL
LIN {X 0,Y 481.299,Z 302.116,A -85,B 0,C 180,E1 -6922.026,E2 -6922.026} C_VEL
LIN {X 0,Y 481.118,Z 309.292,A -85,B 0,C 180,E1 -6923.078,E2 -6923.078} C_VEL
LIN {X 0,Y 480.999,Z 314.943,A -85,B 0,C 180,E1 -6924.13,E2 -6924.13} C_VEL
LIN {X 0,Y 480.866,Z 320.196,A -85,B 0,C 180,E1 -6925.39,E2 -6925.39} C_VEL
LIN {X 0,Y 480.924,Z 322.896,A -85,B 0,C 180,E1 -6926.23,E2 -6926.23} C_VEL
LIN {X 0,Y 480.848,Z 325.849,A -85,B 0,C 180,E1 -6927.487,E2 -6927.487} C_VEL
LIN {X 0,Y 480.822,Z 327.128,A -85,B 0,C 180,E1 -6928.325,E2 -6928.325} C_VEL
LIN {X 0,Y 480.762,Z 327.923,A -85,B 0,C 180,E1 -6929.163,E2 -6929.163} C_VEL
LIN {X 0,Y 480.75,Z 328.23,A -85,B 0,C 180,E1 -6930,E2 -6930} C_VEL
LIN {X 0,Y 480.762,Z 327.941,A -85,B 0,C 180,E1 -6930.838,E2 -6930.838} C_VEL
LIN {X 0,Y 480.822,Z 327.158,A -85,B 0,C 180,E1 -6931.675,E2 -6931.675} C_VEL
LIN {X 0,Y 480.848,Z 325.891,A -85,B 0,C 180,E1 -6932.513,E2 -6932.513} C_VEL
LIN {X 0,Y 480.924,Z 322.964,A -85,B 0,C 180,E1 -6933.771,E2 -6933.771} C_VEL
LIN {X 0,Y 480.866,Z 320.278,A -85,B 0,C 180,E1 -6934.611,E2 -6934.611} C_VEL
LIN {X 0,Y 480.989,Z 316.973,A -85,B 0,C 180,E1 -6935.45,E2 -6935.45} C_VEL
LIN {X 0,Y 481.084,Z 311.274,A -85,B 0,C 180,E1 -6936.59,E2 -6936.59} C_VEL
LIN {X 0,Y 481.234,Z 305.256,A -85,B 0,C 180,E1 -6937.553,E2 -6937.553} C_VEL
LIN {X 0,Y 481.495,Z 297.109,A -85,B 0,C 180,E1 -6938.605,E2 -6938.605} C_VEL
LIN {X 0,Y 481.791,Z 287.527,A -85,B 0,C 180,E1 -6939.551,E2 -6939.551} C_VEL
LIN {X 0,Y 482.041,Z 279.57,A -85,B 0,C 180,E1 -6940.182,E2 -6940.182} C_VEL
LIN {X 0,Y 482.25,Z 271.365,A -85,B 0,C 180,E1 -6940.709,E2 -6940.709} C_VEL
LIN {X 0,Y 482.48,Z 263.154,A -85,B 0,C 180,E1 -6941.125,E2 -6941.125} C_VEL
LIN {X 0,Y 481.875,Z 254.77,A -85,B 0,C 180,E1 -6941.466,E2 -6941.466} C_VEL
LIN {X 0,Y 481.071,Z 246.521,A -85,B 0,C 180,E1 -6941.733,E2 -6941.733} C_VEL
LIN {X 0,Y 481.23,Z 235.436,A -85,B 0,C 180,E1 -6945.241,E2 -6945.241} C_VEL
LIN {X 0,Y 481.472,Z 224.591,A -85,B 0,C 180,E1 -6948.732,E2 -6948.732} C_VEL
LIN {X 0,Y 481.762,Z 215.158,A -85,B 0,C 180,E1 -6951.839,E2 -6951.839} C_VEL
LIN {X 0,Y 482.171,Z 204.743,A -85,B 0,C 180,E1 -6955.351,E2 -6955.351} C_VEL
LIN {X 0,Y 482.57,Z 196.395,A -85,B 0,C 180,E1 -6958.25,E2 -6958.25} C_VEL
LIN {X 0,Y 482.883,Z 189.168,A -85,B 0,C 180,E1 -6960.829,E2 -6960.829} C_VEL
LIN {X 0,Y 482.256,Z 184.434,A -85,B 0,C 180,E1 -6962.63,E2 -6962.63} C_VEL
LIN {X 0,Y 481.697,Z 181.299,A -85,B 0,C 180,E1 -6963.922,E2 -6963.922} C_VEL
LIN {X 0,Y 481.629,Z 181.307,A -85,B 0,C 180,E1 -6966.747,E2 -6966.747} C_VEL
LIN {X 0,Y 481.68,Z 181.297,A -85,B 0,C 180,E1 -6969.94,E2 -6969.94} C_VEL
LIN {X 0,Y 481.641,Z 181.302,A -85,B 0,C 180,E1 -6973.3,E2 -6973.3} C_VEL
LIN {X 0,Y 481.656,Z 181.302,A -85,B 0,C 180,E1 -6975.642,E2 -6975.642} C_VEL
LIN {X 0,Y 481.652,Z 181.302,A -85,B 0,C 180,E1 -6978.957,E2 -6978.957} C_VEL
LIN {X 0,Y 481.658,Z 181.304,A -85,B 0,C 180,E1 -6981.993,E2 -6981.993} C_VEL
LIN {X 0,Y 481.692,Z 181.295,A -85,B 0,C 180,E1 -6985.318,E2 -6985.318} C_VEL
LIN {X 0,Y 481.649,Z 181.304,A -85,B 0,C 180,E1 -6988.311,E2 -6988.311} C_VEL
LIN {X 0,Y 481.702,Z 181.296,A -85,B 0,C 180,E1 -6991.218,E2 -6991.218} C_VEL
LIN {X 0,Y 481.694,Z 181.297,A -85,B 0,C 180,E1 -6994.042,E2 -6994.042} C_VEL
LIN {X 0,Y 481.679,Z 181.298,A -85,B 0,C 180,E1 -6996.812,E2 -6996.812} C_VEL
LIN {X 0,Y 481.7,Z 181.296,A -85,B 0,C 180,E1 -6999.502,E2 -6999.502} C_VEL
LIN {X 0,Y 481.697,Z 181.298,A -85,B 0,C 180,E1 -7002.158,E2 -7002.158} C_VEL
LIN {X 0,Y 481.748,Z 181.29,A -85,B 0,C 180,E1 -7004.775,E2 -7004.775} C_VEL
LIN {X 0,Y 481.755,Z 181.289,A -85,B 0,C 180,E1 -7008.215,E2 -7008.215} C_VEL
LIN {X 0,Y 481.744,Z 181.291,A -85,B 0,C 180,E1 -7011.611,E2 -7011.611} C_VEL
LIN {X 0,Y 481.81,Z 181.281,A -85,B 0,C 180,E1 -7014.139,E2 -7014.139} C_VEL
LIN {X 0,Y 481.929,Z 181.27,A -85,B 0,C 180,E1 -7017.492,E2 -7017.492} C_VEL
LIN {X 0,Y 481.944,Z 181.266,A -85,B 0,C 180,E1 -7019.999,E2 -7019.999} C_VEL
LIN {X 0,Y 481.929,Z 181.266,A -85,B 0,C 180,E1 -7022.507,E2 -7022.507} C_VEL
LIN {X 0,Y 481.809,Z 181.28,A -85,B 0,C 180,E1 -7025.86,E2 -7025.86} C_VEL
LIN {X 0,Y 481.742,Z 181.291,A -85,B 0,C 180,E1 -7028.388,E2 -7028.388} C_VEL
LIN {X 0,Y 481.753,Z 181.289,A -85,B 0,C 180,E1 -7031.784,E2 -7031.784} C_VEL
LIN {X 0,Y 481.744,Z 181.292,A -85,B 0,C 180,E1 -7035.223,E2 -7035.223} C_VEL
LIN {X 0,Y 481.709,Z 181.295,A -85,B 0,C 180,E1 -7038.721,E2 -7038.721} C_VEL
LIN {X 0,Y 481.646,Z 181.302,A -85,B 0,C 180,E1 -7041.394,E2 -7041.394} C_VEL
LIN {X 0,Y 481.661,Z 181.301,A -85,B 0,C 180,E1 -7044.113,E2 -7044.113} C_VEL
LIN {X 0,Y 481.747,Z 181.29,A -85,B 0,C 180,E1 -7047.138,E2 -7047.138} C_VEL
LIN {X 0,Y 481.678,Z 181.3,A -85,B 0,C 180,E1 -7049.74,E2 -7049.74} C_VEL
LIN {X 0,Y 481.671,Z 181.299,A -85,B 0,C 180,E1 -7052.673,E2 -7052.673} C_VEL
LIN {X 0,Y 481.64,Z 181.303,A -85,B 0,C 180,E1 -7055.708,E2 -7055.708} C_VEL
LIN {X 0,Y 481.667,Z 181.298,A -85,B 0,C 180,E1 -7058.858,E2 -7058.858} C_VEL
LIN {X 0,Y 481.649,Z 181.303,A -85,B 0,C 180,E1 -7061.912,E2 -7061.912} C_VEL
LIN {X 0,Y 481.655,Z 181.302,A -85,B 0,C 180,E1 -7064.456,E2 -7064.456} C_VEL
LIN {X 0,Y 481.643,Z 181.304,A -85,B 0,C 180,E1 -7067.838,E2 -7067.838} C_VEL
LIN {X 0,Y 481.674,Z 181.298,A -85,B 0,C 180,E1 -7070.65,E2 -7070.65} C_VEL
LIN {X 0,Y 481.626,Z 181.305,A -85,B 0,C 180,E1 -7073.375,E2 -7073.375} C_VEL
LIN {X 0,Y 481.703,Z 181.296,A -85,B 0,C 180,E1 -7076.329,E2 -7076.329} C_VEL
LIN {X 0,Y 481.652,Z 181.302,A -85,B 0,C 180,E1 -7079.415,E2 -7079.415} C_VEL
LIN {X 0,Y 481.694,Z 181.296,A -85,B 0,C 180,E1 -7082.167,E2 -7082.167} C_VEL
LIN {X 0,Y 481.711,Z 181.294,A -85,B 0,C 180,E1 -7084.969,E2 -7084.969} C_VEL
LIN {X 0,Y 481.631,Z 181.304,A -85,B 0,C 180,E1 -7087.977,E2 -7087.977} C_VEL
LIN {X 0,Y 480.962,Z 181.387,A -85,B 0,C 180,E1 -7088.675,E2 -7088.675} C_VEL
LIN {X 0,Y 478.134,Z 181.74,A -85,B 0,C 180,E1 -7089.809,E2 -7089.809} C_VEL
LIN {X 0,Y 475.749,Z 182.038,A -85,B 0,C 180,E1 -7090.724,E2 -7090.724} C_VEL
LIN {X 0,Y 474.729,Z 182.166,A -85,B 0,C 180,E1 -7091.43,E2 -7091.43} C_VEL
LIN {X 0,Y 474.647,Z 182.174,A -85,B 0,C 180,E1 -7091.668,E2 -7091.668} C_VEL
LIN {X 0,Y 474.692,Z 182.17,A -85,B 0,C 180,E1 -7094.544,E2 -7094.544} C_VEL
LIN {X 0,Y 474.73,Z 182.164,A -85,B 0,C 180,E1 -7098.038,E2 -7098.038} C_VEL
LIN {X 0,Y 474.72,Z 182.166,A -85,B 0,C 180,E1 -7101.486,E2 -7101.486} C_VEL
LIN {X 0,Y 474.77,Z 182.157,A -85,B 0,C 180,E1 -7104.052,E2 -7104.052} C_VEL
LIN {X 0,Y 474.884,Z 182.144,A -85,B 0,C 180,E1 -7107.455,E2 -7107.455} C_VEL
LIN {X 0,Y 474.9,Z 182.143,A -85,B 0,C 180,E1 -7110,E2 -7110} C_VEL
LIN {X 0,Y 474.886,Z 182.145,A -85,B 0,C 180,E1 -7112.545,E2 -7112.545} C_VEL
LIN {X 0,Y 474.771,Z 182.159,A -85,B 0,C 180,E1 -7115.948,E2 -7115.948} C_VEL
LIN {X 0,Y 474.72,Z 182.168,A -85,B 0,C 180,E1 -7118.514,E2 -7118.514} C_VEL
LIN {X 0,Y 474.678,Z 182.17,A -85,B 0,C 180,E1 -7121.963,E2 -7121.963} C_VEL
LIN {X 0,Y 474.389,Z 182.299,A -85,B 0,C 180,E1 -7124.806,E2 -7124.806} C_VEL
LIN {X 0,Y 474.253,Z 187.349,A -85,B 0,C 180,E1 -7128.132,E2 -7128.132} C_VEL
LIN {X 0,Y 474.181,Z 191.729,A -85,B 0,C 180,E1 -7130.977,E2 -7130.977} C_VEL
LIN {X 0,Y 474.061,Z 195.803,A -85,B 0,C 180,E1 -7133.595,E2 -7133.595} C_VEL
LIN {X 0,Y 473.974,Z 200.242,A -85,B 0,C 180,E1 -7136.413,E2 -7136.413} C_VEL
LIN {X 0,Y 473.873,Z 204.858,A -85,B 0,C 180,E1 -7139.303,E2 -7139.303} C_VEL
LIN {X 0,Y 473.842,Z 209.686,A -85,B 0,C 180,E1 -7142.285,E2 -7142.285} C_VEL
LIN {X 0,Y 473.837,Z 212.569,A -85,B 0,C 180,E1 -7144.048,E2 -7144.048} C_VEL
LIN {X 0,Y 475.495,Z 223.178,A -85,B 0,C 180,E1 -7144.491,E2 -7144.491} C_VEL
LIN {X 0,Y 475.407,Z 232.013,A -85,B 0,C 180,E1 -7144.949,E2 -7144.949} C_VEL
LIN {X 0,Y 475.142,Z 241.137,A -85,B 0,C 180,E1 -7145.56,E2 -7145.56} C_VEL
LIN {X 0,Y 474.874,Z 249.65,A -85,B 0,C 180,E1 -7146.298,E2 -7146.298} C_VEL
LIN {X 0,Y 474.606,Z 257.147,A -85,B 0,C 180,E1 -7147.12,E2 -7147.12} C_VEL
LIN {X 0,Y 474.382,Z 263.262,A -85,B 0,C 180,E1 -7147.939,E2 -7147.939} C_VEL
LIN {X 0,Y 474.232,Z 268.304,A -85,B 0,C 180,E1 -7148.757,E2 -7148.757} C_VEL
LIN {X 0,Y 474.059,Z 272.63,A -85,B 0,C 180,E1 -7149.604,E2 -7149.604} C_VEL
LIN {X 0,Y 473.965,Z 276.142,A -85,B 0,C 180,E1 -7150.446,E2 -7150.446} C_VEL
LIN {X 0,Y 473.806,Z 280.576,A -85,B 0,C 180,E1 -7151.873,E2 -7151.873} C_VEL
LIN {X 0,Y 473.762,Z 282.906,A -85,B 0,C 180,E1 -7153.03,E2 -7153.03} C_VEL
LIN {X 0,Y 473.704,Z 284.31,A -85,B 0,C 180,E1 -7154.592,E2 -7154.592} C_VEL
LIN {X 0,Y 473.713,Z 284.227,A -85,B 0,C 180,E1 -7155.791,E2 -7155.791} C_VEL
LIN {X 0,Y 473.754,Z 283.12,A -85,B 0,C 180,E1 -7156.97,E2 -7156.97} C_VEL
LIN {X 0,Y 473.804,Z 280.96,A -85,B 0,C 180,E1 -7158.128,E2 -7158.128} C_VEL
LIN {X 0,Y 473.918,Z 277.687,A -85,B 0,C 180,E1 -7159.271,E2 -7159.271} C_VEL
LIN {X 0,Y 474.07,Z 273.136,A -85,B 0,C 180,E1 -7160.434,E2 -7160.434} C_VEL
LIN {X 0,Y 474.296,Z 267.652,A -85,B 0,C 180,E1 -7161.514,E2 -7161.514} C_VEL
LIN {X 0,Y 474.518,Z 260.459,A -85,B 0,C 180,E1 -7162.611,E2 -7162.611} C_VEL
LIN {X 0,Y 474.772,Z 253.946,A -85,B 0,C 180,E1 -7163.397,E2 -7163.397} C_VEL
LIN {X 0,Y 474.974,Z 246.814,A -85,B 0,C 180,E1 -7164.106,E2 -7164.106} C_VEL
LIN {X 0,Y 475.234,Z 238.41,A -85,B 0,C 180,E1 -7164.779,E2 -7164.779} C_VEL
LIN {X 0,Y 475.547,Z 228.662,A -85,B 0,C 180,E1 -7165.386,E2 -7165.386} C_VEL
LIN {X 0,Y 475.421,Z 222.209,A -85,B 0,C 180,E1 -7165.697,E2 -7165.697} C_VEL
LIN {X 0,Y 473.893,Z 212.984,A -85,B 0,C 180,E1 -7166.094,E2 -7166.094} C_VEL
LIN {X 0,Y 473.931,Z 207.211,A -85,B 0,C 180,E1 -7169.723,E2 -7169.723} C_VEL
LIN {X 0,Y 474.04,Z 202.365,A -85,B 0,C 180,E1 -7172.816,E2 -7172.816} C_VEL
LIN {X 0,Y 474.093,Z 198.244,A -85,B 0,C 180,E1 -7175.477,E2 -7175.477} C_VEL
LIN {X 0,Y 474.176,Z 194,A -85,B 0,C 180,E1 -7178.252,E2 -7178.252} C_VEL
LIN {X 0,Y 474.348,Z 189.094,A -85,B 0,C 180,E1 -7181.483,E2 -7181.483} C_VEL
LIN {X 0,Y 474.447,Z 184.55,A -85,B 0,C 180,E1 -7184.537,E2 -7184.537} C_VEL
LIN {X 0,Y 474.468,Z 182.202,A -85,B 0,C 180,E1 -7186.291,E2 -7186.291} C_VEL
LIN {X 0,Y 474.686,Z 182.173,A -85,B 0,C 180,E1 -7188.038,E2 -7188.038} C_VEL
LIN {X 0,Y 474.729,Z 182.167,A -85,B 0,C 180,E1 -7191.487,E2 -7191.487} C_VEL
LIN {X 0,Y 474.779,Z 182.162,A -85,B 0,C 180,E1 -7194.053,E2 -7194.053} C_VEL
LIN {X 0,Y 474.895,Z 182.145,A -85,B 0,C 180,E1 -7197.456,E2 -7197.456} C_VEL
LIN {X 0,Y 474.913,Z 182.143,A -85,B 0,C 180,E1 -7200.001,E2 -7200.001} C_VEL
LIN {X 0,Y 474.894,Z 182.145,A -85,B 0,C 180,E1 -7202.545,E2 -7202.545} C_VEL
LIN {X 0,Y 474.78,Z 182.16,A -85,B 0,C 180,E1 -7205.948,E2 -7205.948} C_VEL
LIN {X 0,Y 474.715,Z 182.167,A -85,B 0,C 180,E1 -7208.514,E2 -7208.514} C_VEL
LIN {X 0,Y 474.707,Z 182.168,A -85,B 0,C 180,E1 -7211.963,E2 -7211.963} C_VEL
LIN {X 0,Y 474.703,Z 182.168,A -85,B 0,C 180,E1 -7215.456,E2 -7215.456} C_VEL
LIN {X 0,Y 474.668,Z 182.172,A -85,B 0,C 180,E1 -7219.011,E2 -7219.011} C_VEL
LIN {X 0,Y 474.591,Z 182.183,A -85,B 0,C 180,E1 -7221.729,E2 -7221.729} C_VEL
LIN {X 0,Y 474.643,Z 182.175,A -85,B 0,C 180,E1 -7224.494,E2 -7224.494} C_VEL
LIN {X 0,Y 474.684,Z 182.17,A -85,B 0,C 180,E1 -7227.335,E2 -7227.335} C_VEL
LIN {X 0,Y 474.608,Z 182.18,A -85,B 0,C 180,E1 -7230.23,E2 -7230.23} C_VEL
LIN {X 0,Y 474.645,Z 182.175,A -85,B 0,C 180,E1 -7233.22,E2 -7233.22} C_VEL
LIN {X 0,Y 474.591,Z 182.181,A -85,B 0,C 180,E1 -7236.324,E2 -7236.324} C_VEL
LIN {X 0,Y 474.62,Z 182.179,A -85,B 0,C 180,E1 -7239.646,E2 -7239.646} C_VEL
LIN {X 0,Y 474.617,Z 182.181,A -85,B 0,C 180,E1 -7242.934,E2 -7242.934} C_VEL
LIN {X 0,Y 474.611,Z 182.183,A -85,B 0,C 180,E1 -7245.895,E2 -7245.895} C_VEL
LIN {X 0,Y 474.629,Z 182.178,A -85,B 0,C 180,E1 -7249.041,E2 -7249.041} C_VEL
LIN {X 0,Y 474.612,Z 182.181,A -85,B 0,C 180,E1 -7251.704,E2 -7251.704} C_VEL
LIN {X 0,Y 474.657,Z 182.182,A -85,B 0,C 180,E1 -7255.246,E2 -7255.246} C_VEL
LIN {X 0,Y 474.71,Z 182.284,A -85,B 0,C 180,E1 -7255.637,E2 -7255.637} C_VEL
LIN {X 0,Y 475.81,Z 188.784,A -85,B 0,C 180,E1 -7258.375,E2 -7258.375} C_VEL
LIN {X 0,Y 475.814,Z 193.758,A -85,B 0,C 180,E1 -7260.301,E2 -7260.301} C_VEL
LIN {X 0,Y 475.208,Z 202.852,A -85,B 0,C 180,E1 -7263.661,E2 -7263.661} C_VEL
LIN {X 0,Y 474.815,Z 211.138,A -85,B 0,C 180,E1 -7266.592,E2 -7266.592} C_VEL
LIN {X 0,Y 474.524,Z 220.049,A -85,B 0,C 180,E1 -7269.632,E2 -7269.632} C_VEL
LIN {X 0,Y 474.313,Z 228.09,A -85,B 0,C 180,E1 -7272.317,E2 -7272.317} C_VEL
LIN {X 0,Y 474.075,Z 237.579,A -85,B 0,C 180,E1 -7275.403,E2 -7275.403} C_VEL
LIN {X 0,Y 474.004,Z 245.967,A -85,B 0,C 180,E1 -7278.096,E2 -7278.096} C_VEL
LIN {X 0,Y 475.19,Z 258.334,A -85,B 0,C 180,E1 -7278.508,E2 -7278.508} C_VEL
LIN {X 0,Y 475.4,Z 265.402,A -85,B 0,C 180,E1 -7278.83,E2 -7278.83} C_VEL
LIN {X 0,Y 475.107,Z 276.069,A -85,B 0,C 180,E1 -7279.452,E2 -7279.452} C_VEL
LIN {X 0,Y 474.811,Z 284.556,A -85,B 0,C 180,E1 -7280.092,E2 -7280.092} C_VEL
LIN {X 0,Y 474.547,Z 292.572,A -85,B 0,C 180,E1 -7280.839,E2 -7280.839} C_VEL
LIN {X 0,Y 474.367,Z 298.343,A -85,B 0,C 180,E1 -7281.48,E2 -7281.48} C_VEL
LIN {X 0,Y 474.168,Z 304.788,A -85,B 0,C 180,E1 -7282.334,E2 -7282.334} C_VEL
LIN {X 0,Y 474.028,Z 311.263,A -85,B 0,C 180,E1 -7283.39,E2 -7283.39} C_VEL
LIN {X 0,Y 473.904,Z 316.55,A -85,B 0,C 180,E1 -7284.469,E2 -7284.469} C_VEL
LIN {X 0,Y 473.755,Z 321.374,A -85,B 0,C 180,E1 -7285.746,E2 -7285.746} C_VEL
LIN {X 0,Y 473.844,Z 323.741,A -85,B 0,C 180,E1 -7286.599,E2 -7286.599} C_VEL
LIN {X 0,Y 473.765,Z 325.524,A -85,B 0,C 180,E1 -7287.449,E2 -7287.449} C_VEL
LIN {X 0,Y 473.755,Z 326.804,A -85,B 0,C 180,E1 -7288.3,E2 -7288.3} C_VEL
LIN {X 0,Y 473.691,Z 327.599,A -85,B 0,C 180,E1 -7289.15,E2 -7289.15} C_VEL
LIN {X 0,Y 473.676,Z 327.905,A -85,B 0,C 180,E1 -7290,E2 -7290} C_VEL
LIN {X 0,Y 473.69,Z 327.617,A -85,B 0,C 180,E1 -7290.85,E2 -7290.85} C_VEL
LIN {X 0,Y 473.755,Z 326.831,A -85,B 0,C 180,E1 -7291.7,E2 -7291.7} C_VEL
LIN {X 0,Y 473.765,Z 325.561,A -85,B 0,C 180,E1 -7292.551,E2 -7292.551} C_VEL
LIN {X 0,Y 473.827,Z 322.629,A -85,B 0,C 180,E1 -7293.827,E2 -7293.827} C_VEL
LIN {X 0,Y 473.789,Z 319.938,A -85,B 0,C 180,E1 -7294.68,E2 -7294.68} C_VEL
LIN {X 0,Y 473.904,Z 316.625,A -85,B 0,C 180,E1 -7295.532,E2 -7295.532} C_VEL
LIN {X 0,Y 474.008,Z 311.467,A -85,B 0,C 180,E1 -7296.589,E2 -7296.589} C_VEL
LIN {X 0,Y 474.142,Z 306.312,A -85,B 0,C 180,E1 -7297.452,E2 -7297.452} C_VEL
LIN {X 0,Y 474.318,Z 300.161,A -85,B 0,C 180,E1 -7298.307,E2 -7298.307} C_VEL
LIN {X 0,Y 474.539,Z 293.7,A -85,B 0,C 180,E1 -7299.054,E2 -7299.054} C_VEL
LIN {X 0,Y 474.774,Z 285.874,A -85,B 0,C 180,E1 -7299.802,E2 -7299.802} C_VEL
LIN {X 0,Y 475.071,Z 277.626,A -85,B 0,C 180,E1 -7300.441,E2 -7300.441} C_VEL
LIN {X 0,Y 475.386,Z 267.148,A -85,B 0,C 180,E1 -7301.081,E2 -7301.081} C_VEL
LIN {X 0,Y 475.301,Z 259.268,A -85,B 0,C 180,E1 -7301.445,E2 -7301.445} C_VEL
LIN {X 0,Y 474.03,Z 246.807,A -85,B 0,C 180,E1 -7301.87,E2 -7301.87} C_VEL
LIN {X 0,Y 473.984,Z 246.199,A -85,B 0,C 180,E1 -7301.917,E2 -7301.917} C_VEL
LIN {X 0,Y 474.183,Z 234.931,A -85,B 0,C 180,E1 -7305.552,E2 -7305.552} C_VEL
LIN {X 0,Y 474.437,Z 224.404,A -85,B 0,C 180,E1 -7309.02,E2 -7309.02} C_VEL
LIN {X 0,Y 474.749,Z 214.982,A -85,B 0,C 180,E1 -7312.179,E2 -7312.179} C_VEL
LIN {X 0,Y 475.2,Z 204.198,A -85,B 0,C 180,E1 -7315.893,E2 -7315.893} C_VEL
LIN {X 0,Y 475.67,Z 194.933,A -85,B 0,C 180,E1 -7319.181,E2 -7319.181} C_VEL
LIN {X 0,Y 475.869,Z 189.621,A -85,B 0,C 180,E1 -7321.125,E2 -7321.125} C_VEL
LIN {X 0,Y 474.669,Z 182.174,A -85,B 0,C 180,E1 -7324.075,E2 -7324.075} C_VEL
LIN {X 0,Y 474.593,Z 182.182,A -85,B 0,C 180,E1 -7327.384,E2 -7327.384} C_VEL
LIN {X 0,Y 474.62,Z 182.179,A -85,B 0,C 180,E1 -7330.658,E2 -7330.658} C_VEL
LIN {X 0,Y 474.604,Z 182.178,A -85,B 0,C 180,E1 -7333.481,E2 -7333.481} C_VEL
LIN {X 0,Y 474.595,Z 182.182,A -85,B 0,C 180,E1 -7336.52,E2 -7336.52} C_VEL
LIN {X 0,Y 474.618,Z 182.178,A -85,B 0,C 180,E1 -7339.342,E2 -7339.342} C_VEL
LIN {X 0,Y 474.594,Z 182.181,A -85,B 0,C 180,E1 -7342.616,E2 -7342.616} C_VEL
LIN {X 0,Y 474.636,Z 182.177,A -85,B 0,C 180,E1 -7345.759,E2 -7345.759} C_VEL
LIN {X 0,Y 474.603,Z 182.178,A -85,B 0,C 180,E1 -7348.782,E2 -7348.782} C_VEL
LIN {X 0,Y 474.648,Z 182.175,A -85,B 0,C 180,E1 -7351.717,E2 -7351.717} C_VEL
LIN {X 0,Y 474.656,Z 182.174,A -85,B 0,C 180,E1 -7354.582,E2 -7354.582} C_VEL
LIN {X 0,Y 474.605,Z 182.181,A -85,B 0,C 180,E1 -7357.355,E2 -7357.355} C_VEL
LIN {X 0,Y 474.659,Z 182.173,A -85,B 0,C 180,E1 -7360.089,E2 -7360.089} C_VEL
LIN {X 0,Y 474.643,Z 182.174,A -85,B 0,C 180,E1 -7362.774,E2 -7362.774} C_VEL
LIN {X 0,Y 474.653,Z 182.174,A -85,B 0,C 180,E1 -7365.421,E2 -7365.421} C_VEL
LIN {X 0,Y 474.709,Z 182.166,A -85,B 0,C 180,E1 -7368.037,E2 -7368.037} C_VEL
LIN {X 0,Y 474.715,Z 182.167,A -85,B 0,C 180,E1 -7371.486,E2 -7371.486} C_VEL
LIN {X 0,Y 474.772,Z 182.158,A -85,B 0,C 180,E1 -7374.052,E2 -7374.052} C_VEL
LIN {X 0,Y 474.895,Z 182.146,A -85,B 0,C 180,E1 -7377.455,E2 -7377.455} C_VEL
LIN {X 0,Y 474.915,Z 182.141,A -85,B 0,C 180,E1 -7379.999,E2 -7379.999} C_VEL
LIN {X 0,Y 474.896,Z 182.143,A -85,B 0,C 180,E1 -7382.544,E2 -7382.544} C_VEL
LIN {X 0,Y 474.772,Z 182.157,A -85,B 0,C 180,E1 -7385.947,E2 -7385.947} C_VEL
LIN {X 0,Y 474.714,Z 182.166,A -85,B 0,C 180,E1 -7388.513,E2 -7388.513} C_VEL
LIN {X 0,Y 474.707,Z 182.167,A -85,B 0,C 180,E1 -7391.961,E2 -7391.961} C_VEL
LIN {X 0,Y 474.701,Z 182.168,A -85,B 0,C 180,E1 -7395.455,E2 -7395.455} C_VEL
LIN {X 0,Y 474.664,Z 182.174,A -85,B 0,C 180,E1 -7399.009,E2 -7399.009} C_VEL
LIN {X 0,Y 474.589,Z 182.181,A -85,B 0,C 180,E1 -7401.728,E2 -7401.728} C_VEL
LIN {X 0,Y 474.64,Z 182.178,A -85,B 0,C 180,E1 -7404.493,E2 -7404.493} C_VEL
LIN {X 0,Y 474.699,Z 182.167,A -85,B 0,C 180,E1 -7407.338,E2 -7407.338} C_VEL
LIN {X 0,Y 474.603,Z 182.181,A -85,B 0,C 180,E1 -7410.809,E2 -7410.809} C_VEL
LIN {X 0,Y 474.636,Z 182.176,A -85,B 0,C 180,E1 -7413.983,E2 -7413.983} C_VEL
LIN {X 0,Y 474.572,Z 182.185,A -85,B 0,C 180,E1 -7416.899,E2 -7416.899} C_VEL
LIN {X 0,Y 474.624,Z 182.177,A -85,B 0,C 180,E1 -7419.646,E2 -7419.646} C_VEL
LIN {X 0,Y 474.611,Z 182.177,A -85,B 0,C 180,E1 -7422.933,E2 -7422.933} C_VEL
LIN {X 0,Y 474.604,Z 182.181,A -85,B 0,C 180,E1 -7425.894,E2 -7425.894} C_VEL
LIN {X 0,Y 474.623,Z 182.178,A -85,B 0,C 180,E1 -7429.04,E2 -7429.04} C_VEL
LIN {X 0,Y 474.605,Z 182.18,A -85,B 0,C 180,E1 -7431.703,E2 -7431.703} C_VEL
LIN {X 0,Y 474.625,Z 182.176,A -85,B 0,C 180,E1 -7434.725,E2 -7434.725} C_VEL
LIN {X 0,Y 474.632,Z 182.178,A -85,B 0,C 180,E1 -7437.787,E2 -7437.787} C_VEL
LIN {X 0,Y 474.625,Z 182.176,A -85,B 0,C 180,E1 -7440.882,E2 -7440.882} C_VEL
LIN {X 0,Y 474.653,Z 182.174,A -85,B 0,C 180,E1 -7443.628,E2 -7443.628} C_VEL
LIN {X 0,Y 474.628,Z 182.177,A -85,B 0,C 180,E1 -7446.64,E2 -7446.64} C_VEL
LIN {X 0,Y 474.649,Z 182.175,A -85,B 0,C 180,E1 -7450.089,E2 -7450.089} C_VEL
LIN {X 0,Y 474.647,Z 182.174,A -85,B 0,C 180,E1 -7451.668,E2 -7451.668} C_VEL
LIN {X 0,Y 473.984,Z 182.257,A -85,B 0,C 180,E1 -7452.377,E2 -7452.377} C_VEL
LIN {X 0,Y 471.133,Z 182.615,A -85,B 0,C 180,E1 -7453.529,E2 -7453.529} C_VEL
LIN {X 0,Y 468.719,Z 182.916,A -85,B 0,C 180,E1 -7454.457,E2 -7454.457} C_VEL
LIN {X 0,Y 467.68,Z 183.043,A -85,B 0,C 180,E1 -7455.175,E2 -7455.175} C_VEL
LIN {X 0,Y 467.594,Z 183.052,A -85,B 0,C 180,E1 -7455.417,E2 -7455.417} C_VEL
LIN {X 0,Y 467.688,Z 183.042,A -85,B 0,C 180,E1 -7457.855,E2 -7457.855} C_VEL
LIN {X 0,Y 467.674,Z 183.043,A -85,B 0,C 180,E1 -7461.357,E2 -7461.357} C_VEL
LIN {X 0,Y 467.735,Z 183.034,A -85,B 0,C 180,E1 -7463.962,E2 -7463.962} C_VEL
LIN {X 0,Y 467.849,Z 183.02,A -85,B 0,C 180,E1 -7467.417,E2 -7467.417} C_VEL
LIN {X 0,Y 467.871,Z 183.019,A -85,B 0,C 180,E1 -7470,E2 -7470} C_VEL
LIN {X 0,Y 467.852,Z 183.022,A -85,B 0,C 180,E1 -7472.583,E2 -7472.583} C_VEL
LIN {X 0,Y 467.735,Z 183.036,A -85,B 0,C 180,E1 -7476.037,E2 -7476.037} C_VEL
LIN {X 0,Y 467.673,Z 183.045,A -85,B 0,C 180,E1 -7478.643,E2 -7478.643} C_VEL
LIN {X 0,Y 467.627,Z 183.049,A -85,B 0,C 180,E1 -7482.146,E2 -7482.146} C_VEL
LIN {X 0,Y 467.341,Z 183.114,A -85,B 0,C 180,E1 -7484.812,E2 -7484.812} C_VEL
LIN {X 0,Y 467.188,Z 187.155,A -85,B 0,C 180,E1 -7487.509,E2 -7487.509} C_VEL
LIN {X 0,Y 467.095,Z 191.326,A -85,B 0,C 180,E1 -7490.247,E2 -7490.247} C_VEL
LIN {X 0,Y 467.008,Z 196.135,A -85,B 0,C 180,E1 -7493.369,E2 -7493.369} C_VEL
LIN {X 0,Y 466.927,Z 200.039,A -85,B 0,C 180,E1 -7495.88,E2 -7495.88} C_VEL
LIN {X 0,Y 466.807,Z 204.666,A -85,B 0,C 180,E1 -7498.801,E2 -7498.801} C_VEL
LIN {X 0,Y 466.762,Z 209.45,A -85,B 0,C 180,E1 -7501.802,E2 -7501.802} C_VEL
LIN {X 0,Y 466.746,Z 212.793,A -85,B 0,C 180,E1 -7503.879,E2 -7503.879} C_VEL
LIN {X 0,Y 468.404,Z 223.309,A -85,B 0,C 180,E1 -7504.326,E2 -7504.326} C_VEL
LIN {X 0,Y 468.471,Z 230.168,A -85,B 0,C 180,E1 -7504.676,E2 -7504.676} C_VEL
LIN {X 0,Y 468.225,Z 237.956,A -85,B 0,C 180,E1 -7505.17,E2 -7505.17} C_VEL
LIN {X 0,Y 467.952,Z 246.505,A -85,B 0,C 180,E1 -7505.854,E2 -7505.854} C_VEL
LIN {X 0,Y 467.721,Z 254.696,A -85,B 0,C 180,E1 -7506.676,E2 -7506.676} C_VEL
LIN {X 0,Y 467.403,Z 261.964,A -85,B 0,C 180,E1 -7507.594,E2 -7507.594} C_VEL
LIN {X 0,Y 467.22,Z 267.919,A -85,B 0,C 180,E1 -7508.54,E2 -7508.54} C_VEL
LIN {X 0,Y 467.009,Z 272.936,A -85,B 0,C 180,E1 -7509.527,E2 -7509.527} C_VEL
LIN {X 0,Y 466.851,Z 277.754,A -85,B 0,C 180,E1 -7510.75,E2 -7510.75} C_VEL
LIN {X 0,Y 466.736,Z 281.24,A -85,B 0,C 180,E1 -7511.966,E2 -7511.966} C_VEL
LIN {X 0,Y 466.676,Z 282.604,A -85,B 0,C 180,E1 -7512.663,E2 -7512.663} C_VEL
LIN {X 0,Y 466.649,Z 284.215,A -85,B 0,C 180,E1 -7513.851,E2 -7513.851} C_VEL
LIN {X 0,Y 466.621,Z 284.792,A -85,B 0,C 180,E1 -7515.063,E2 -7515.063} C_VEL
LIN {X 0,Y 466.655,Z 284.228,A -85,B 0,C 180,E1 -7516.294,E2 -7516.294} C_VEL
LIN {X 0,Y 466.677,Z 282.51,A -85,B 0,C 180,E1 -7517.555,E2 -7517.555} C_VEL
LIN {X 0,Y 466.758,Z 280.426,A -85,B 0,C 180,E1 -7518.51,E2 -7518.51} C_VEL
LIN {X 0,Y 466.897,Z 276.885,A -85,B 0,C 180,E1 -7519.666,E2 -7519.666} C_VEL
LIN {X 0,Y 467.082,Z 272.216,A -85,B 0,C 180,E1 -7520.807,E2 -7520.807} C_VEL
LIN {X 0,Y 467.317,Z 266.148,A -85,B 0,C 180,E1 -7521.933,E2 -7521.933} C_VEL
LIN {X 0,Y 467.536,Z 260.14,A -85,B 0,C 180,E1 -7522.816,E2 -7522.816} C_VEL
LIN {X 0,Y 467.793,Z 253.637,A -85,B 0,C 180,E1 -7523.6,E2 -7523.6} C_VEL
LIN {X 0,Y 468.048,Z 245.981,A -85,B 0,C 180,E1 -7524.355,E2 -7524.355} C_VEL
LIN {X 0,Y 468.292,Z 238.28,A -85,B 0,C 180,E1 -7524.969,E2 -7524.969} C_VEL
LIN {X 0,Y 468.619,Z 228.628,A -85,B 0,C 180,E1 -7525.573,E2 -7525.573} C_VEL
LIN {X 0,Y 468.458,Z 222.952,A -85,B 0,C 180,E1 -7525.85,E2 -7525.85} C_VEL
LIN {X 0,Y 466.799,Z 213.27,A -85,B 0,C 180,E1 -7526.278,E2 -7526.278} C_VEL
LIN {X 0,Y 466.832,Z 208.659,A -85,B 0,C 180,E1 -7529.214,E2 -7529.214} C_VEL
LIN {X 0,Y 466.976,Z 203.363,A -85,B 0,C 180,E1 -7532.617,E2 -7532.617} C_VEL
LIN {X 0,Y 467.051,Z 198.159,A -85,B 0,C 180,E1 -7536.029,E2 -7536.029} C_VEL
LIN {X 0,Y 467.153,Z 193.875,A -85,B 0,C 180,E1 -7538.867,E2 -7538.867} C_VEL
LIN {X 0,Y 467.301,Z 189.795,A -85,B 0,C 180,E1 -7541.59,E2 -7541.59} C_VEL
LIN {X 0,Y 467.412,Z 185.812,A -85,B 0,C 180,E1 -7544.298,E2 -7544.298} C_VEL
LIN {X 0,Y 467.394,Z 183.231,A -85,B 0,C 180,E1 -7546.08,E2 -7546.08} C_VEL
LIN {X 0,Y 467.636,Z 183.052,A -85,B 0,C 180,E1 -7547.855,E2 -7547.855} C_VEL
LIN {X 0,Y 467.682,Z 183.046,A -85,B 0,C 180,E1 -7551.358,E2 -7551.358} C_VEL
LIN {X 0,Y 467.744,Z 183.039,A -85,B 0,C 180,E1 -7553.963,E2 -7553.963} C_VEL
LIN {X 0,Y 467.86,Z 183.022,A -85,B 0,C 180,E1 -7557.418,E2 -7557.418} C_VEL
LIN {X 0,Y 467.884,Z 183.018,A -85,B 0,C 180,E1 -7560.001,E2 -7560.001} C_VEL
LIN {X 0,Y 467.86,Z 183.021,A -85,B 0,C 180,E1 -7562.584,E2 -7562.584} C_VEL
LIN {X 0,Y 467.744,Z 183.036,A -85,B 0,C 180,E1 -7566.038,E2 -7566.038} C_VEL
LIN {X 0,Y 467.672,Z 183.043,A -85,B 0,C 180,E1 -7568.644,E2 -7568.644} C_VEL
LIN {X 0,Y 467.658,Z 183.045,A -85,B 0,C 180,E1 -7572.146,E2 -7572.146} C_VEL
LIN {X 0,Y 467.642,Z 183.047,A -85,B 0,C 180,E1 -7575.695,E2 -7575.695} C_VEL
LIN {X 0,Y 467.621,Z 183.05,A -85,B 0,C 180,E1 -7578.765,E2 -7578.765} C_VEL
LIN {X 0,Y 467.583,Z 183.055,A -85,B 0,C 180,E1 -7581.269,E2 -7581.269} C_VEL
LIN {X 0,Y 467.566,Z 183.057,A -85,B 0,C 180,E1 -7583.944,E2 -7583.944} C_VEL
LIN {X 0,Y 467.616,Z 183.052,A -85,B 0,C 180,E1 -7586.801,E2 -7586.801} C_VEL
LIN {X 0,Y 467.557,Z 183.059,A -85,B 0,C 180,E1 -7589.738,E2 -7589.738} C_VEL
LIN {X 0,Y 467.586,Z 183.054,A -85,B 0,C 180,E1 -7592.759,E2 -7592.759} C_VEL
LIN {X 0,Y 467.556,Z 183.059,A -85,B 0,C 180,E1 -7595.89,E2 -7595.89} C_VEL
LIN {X 0,Y 467.578,Z 183.058,A -85,B 0,C 180,E1 -7599.146,E2 -7599.146} C_VEL
LIN {X 0,Y 467.589,Z 183.058,A -85,B 0,C 180,E1 -7602.567,E2 -7602.567} C_VEL
LIN {X 0,Y 467.572,Z 183.059,A -85,B 0,C 180,E1 -7605.053,E2 -7605.053} C_VEL
LIN {X 0,Y 467.591,Z 183.056,A -85,B 0,C 180,E1 -7607.44,E2 -7607.44} C_VEL
LIN {X 0,Y 467.584,Z 183.056,A -85,B 0,C 180,E1 -7610.856,E2 -7610.856} C_VEL
LIN {X 0,Y 467.564,Z 183.064,A -85,B 0,C 180,E1 -7614.261,E2 -7614.261} C_VEL
LIN {X 0,Y 467.656,Z 183.23,A -85,B 0,C 180,E1 -7615.414,E2 -7615.414} C_VEL
LIN {X 0,Y 468.835,Z 190.064,A -85,B 0,C 180,E1 -7618.355,E2 -7618.355} C_VEL
LIN {X 0,Y 468.787,Z 195.268,A -85,B 0,C 180,E1 -7620.404,E2 -7620.404} C_VEL
LIN {X 0,Y 468.184,Z 204.069,A -85,B 0,C 180,E1 -7623.716,E2 -7623.716} C_VEL
LIN {X 0,Y 467.737,Z 213.25,A -85,B 0,C 180,E1 -7627.004,E2 -7627.004} C_VEL
LIN {X 0,Y 467.43,Z 222.558,A -85,B 0,C 180,E1 -7630.227,E2 -7630.227} C_VEL
LIN {X 0,Y 467.124,Z 231.93,A -85,B 0,C 180,E1 -7633.39,E2 -7633.39} C_VEL
LIN {X 0,Y 466.902,Z 241.395,A -85,B 0,C 180,E1 -7636.508,E2 -7636.508} C_VEL
LIN {X 0,Y 466.885,Z 245.656,A -85,B 0,C 180,E1 -7637.9,E2 -7637.9} C_VEL
LIN {X 0,Y 468.176,Z 258.611,A -85,B 0,C 180,E1 -7638.36,E2 -7638.36} C_VEL
LIN {X 0,Y 468.424,Z 265.389,A -85,B 0,C 180,E1 -7638.675,E2 -7638.675} C_VEL
LIN {X 0,Y 468.129,Z 275.755,A -85,B 0,C 180,E1 -7639.293,E2 -7639.293} C_VEL
LIN {X 0,Y 467.813,Z 284.241,A -85,B 0,C 180,E1 -7639.942,E2 -7639.942} C_VEL
LIN {X 0,Y 467.496,Z 292.255,A -85,B 0,C 180,E1 -7640.7,E2 -7640.7} C_VEL
LIN {X 0,Y 467.335,Z 298.024,A -85,B 0,C 180,E1 -7641.351,E2 -7641.351} C_VEL
LIN {X 0,Y 467.098,Z 304.466,A -85,B 0,C 180,E1 -7642.218,E2 -7642.218} C_VEL
LIN {X 0,Y 466.953,Z 310.833,A -85,B 0,C 180,E1 -7643.269,E2 -7643.269} C_VEL
LIN {X 0,Y 466.82,Z 316.227,A -85,B 0,C 180,E1 -7644.384,E2 -7644.384} C_VEL
LIN {X 0,Y 466.668,Z 321.05,A -85,B 0,C 180,E1 -7645.682,E2 -7645.682} C_VEL
LIN {X 0,Y 466.756,Z 323.418,A -85,B 0,C 180,E1 -7646.547,E2 -7646.547} C_VEL
LIN {X 0,Y 466.685,Z 325.201,A -85,B 0,C 180,E1 -7647.411,E2 -7647.411} C_VEL
LIN {X 0,Y 466.661,Z 326.48,A -85,B 0,C 180,E1 -7648.274,E2 -7648.274} C_VEL
LIN {X 0,Y 466.622,Z 327.275,A -85,B 0,C 180,E1 -7649.137,E2 -7649.137} C_VEL
LIN {X 0,Y 466.605,Z 327.58,A -85,B 0,C 180,E1 -7650,E2 -7650} C_VEL
LIN {X 0,Y 466.621,Z 327.292,A -85,B 0,C 180,E1 -7650.863,E2 -7650.863} C_VEL
LIN {X 0,Y 466.661,Z 326.502,A -85,B 0,C 180,E1 -7651.726,E2 -7651.726} C_VEL
